C03650=1172.212,-91.528,-41.773,179.063,5.775,149.305
C03651=1172.217,-91.777,-41.762,179.061,5.775,149.306
C03652=1172.222,-92.027,-41.753,179.058,5.775,149.306
C03653=1172.228,-92.276,-41.743,179.057,5.775,149.307
C03654=1172.232,-92.527,-41.733,179.054,5.774,149.307
C03655=1172.238,-92.776,-41.723,179.052,5.773,149.308
C03656=1172.243,-93.026,-41.713,179.050,5.774,149.309
C03657=1172.249,-93.276,-41.704,179.048,5.773,149.309
C03658=1172.254,-93.525,-41.694,179.046,5.773,149.310
C03659=1172.259,-93.774,-41.684,179.043,5.773,149.310
C03660=1172.264,-94.025,-41.674,179.041,5.772,149.311
C03661=1172.270,-94.275,-41.664,179.039,5.772,149.312
C03662=1172.275,-94.524,-41.655,179.036,5.772,149.312
C03663=1172.281,-94.774,-41.645,179.035,5.772,149.313
C03664=1172.286,-95.023,-41.635,179.032,5.771,149.313
C03665=1172.291,-95.273,-41.625,179.030,5.771,149.314
C03666=1172.296,-95.524,-41.615,179.028,5.771,149.315
C03667=1172.301,-95.773,-41.606,179.026,5.770,149.315
C03668=1172.307,-96.023,-41.596,179.024,5.771,149.316
C03669=1172.312,-96.273,-41.587,179.021,5.770,149.316
C03670=1172.318,-96.522,-41.576,179.020,5.770,149.317
C03671=1172.323,-96.772,-41.568,179.017,5.770,149.318
C03672=1172.328,-97.021,-41.557,179.015,5.769,149.318
C03673=1172.333,-97.272,-41.548,179.013,5.769,149.319
C03674=1172.339,-97.522,-41.538,179.011,5.768,149.319
C03675=1172.344,-97.771,-41.529,179.009,5.769,149.320
C03676=1172.349,-98.021,-41.519,179.006,5.768,149.320
C03677=1172.354,-98.271,-41.510,179.004,5.768,149.321
C03678=1172.360,-98.520,-41.500,179.002,5.768,149.322
C03679=1172.365,-98.770,-41.490,179.000,5.767,149.322
C03680=1172.371,-99.020,-41.481,178.998,5.767,149.323
C03681=1172.376,-99.269,-41.471,178.995,5.767,149.323
C03682=1172.381,-99.520,-41.461,178.994,5.767,149.324
C03683=1172.386,-99.769,-41.451,178.991,5.766,149.324
C03684=1172.392,-100.019,-41.442,178.989,5.766,149.325
C03685=1172.397,-100.268,-41.432,178.987,5.766,149.326
C03686=1172.403,-100.519,-41.423,178.985,5.765,149.326
C03687=1172.408,-100.768,-41.414,178.983,5.765,149.327
C03688=1172.413,-101.018,-41.404,178.980,5.765,149.328
C03689=1172.418,-101.268,-41.395,178.979,5.765,149.328
C03690=1172.424,-101.517,-41.385,178.976,5.765,149.329
C03691=1172.430,-101.789,-41.374,178.974,5.764,149.329
C03692=1172.435,-102.061,-41.364,178.972,5.764,149.330
C03693=1172.441,-102.333,-41.354,178.969,5.764,149.331
C03694=1172.447,-102.605,-41.343,178.967,5.763,149.331
C03695=1172.452,-102.854,-41.334,178.965,5.764,149.332
C03696=1172.457,-103.104,-41.325,178.963,5.763,149.332
C03697=1172.463,-103.355,-41.315,178.960,5.762,149.333
C03698=1172.468,-103.604,-41.306,178.958,5.762,149.334
C03699=1172.473,-103.854,-41.296,178.956,5.762,149.334
C03700=1172.478,-104.103,-41.286,178.954,5.762,149.335
C03701=1172.484,-104.353,-41.278,178.952,5.761,149.335
C03702=1172.489,-104.603,-41.268,178.950,5.762,149.336
C03703=1172.494,-104.853,-41.258,178.948,5.761,149.336
C03704=1172.500,-105.103,-41.249,178.945,5.761,149.337
C03705=1172.505,-105.353,-41.240,178.943,5.761,149.338
C03706=1172.510,-105.602,-41.230,178.941,5.760,149.338
C03707=1172.516,-105.852,-41.221,178.939,5.760,149.339
C03708=1172.521,-106.102,-41.212,178.937,5.759,149.339
C03709=1172.526,-106.351,-41.202,178.935,5.760,149.340
C03710=1172.532,-106.601,-41.193,178.933,5.759,149.341
C03711=1172.537,-106.851,-41.184,178.930,5.760,149.341
C03712=1172.542,-107.100,-41.174,178.928,5.759,149.342
C03713=1172.548,-107.350,-41.165,178.927,5.759,149.342
C03714=1172.553,-107.600,-41.156,178.924,5.758,149.343
C03715=1172.558,-107.849,-41.146,178.922,5.758,149.343
C03716=1172.564,-108.100,-41.137,178.920,5.758,149.344
C03717=1172.569,-108.350,-41.128,178.918,5.757,149.345
C03718=1172.574,-108.599,-41.119,178.915,5.758,149.345
C03719=1172.580,-108.849,-41.109,178.913,5.757,149.346
C03720=1172.585,-109.099,-41.100,178.912,5.757,149.346
C03721=1172.590,-109.349,-41.091,178.909,5.757,149.347
C03722=1172.595,-109.598,-41.082,178.907,5.757,149.347
C03723=1172.601,-109.848,-41.072,178.905,5.756,149.348
C03724=1172.606,-110.098,-41.063,178.903,5.756,149.349
C03725=1172.611,-110.348,-41.054,178.901,5.755,149.349
C03726=1172.617,-110.598,-41.045,178.899,5.756,149.350
C03727=1172.622,-110.847,-41.035,178.897,5.755,149.350
C03728=1172.627,-111.097,-41.026,178.894,5.755,149.351
C03729=1172.632,-111.347,-41.017,178.892,5.755,149.352
C03730=1172.638,-111.597,-41.008,178.890,5.754,149.352
C03731=1172.644,-111.846,-40.999,178.888,5.754,149.353
C03732=1172.649,-112.095,-40.990,178.886,5.754,149.353
C03733=1172.654,-112.345,-40.981,178.884,5.754,149.354
C03734=1172.660,-112.595,-40.971,178.882,5.753,149.354
C03735=1172.665,-112.845,-40.962,178.880,5.753,149.355
C03736=1172.670,-113.095,-40.953,178.877,5.753,149.356
C03737=1172.675,-113.345,-40.945,178.876,5.753,149.356
C03738=1172.681,-113.595,-40.935,178.873,5.753,149.357
C03739=1172.686,-113.844,-40.925,178.871,5.753,149.357
C03740=1172.691,-114.094,-40.917,178.869,5.752,149.358
C03741=1172.697,-114.344,-40.908,178.867,5.752,149.359
C03742=1172.702,-114.594,-40.899,178.865,5.751,149.359
C03743=1172.708,-114.843,-40.890,178.863,5.752,149.360
C03744=1172.713,-115.093,-40.881,178.861,5.751,149.360
C03745=1172.719,-115.343,-40.872,178.859,5.751,149.361
C03746=1172.724,-115.593,-40.863,178.856,5.751,149.361
C03747=1172.729,-115.843,-40.854,178.854,5.750,149.362
C03748=1172.735,-116.093,-40.845,178.853,5.750,149.362
C03749=1172.740,-116.342,-40.835,178.850,5.750,149.363
C03750=1172.745,-116.592,-40.826,178.848,5.750,149.364
C03751=1172.750,-116.842,-40.817,178.846,5.749,149.364
C03752=1172.756,-117.091,-40.809,178.844,5.749,149.365
C03753=1172.761,-117.341,-40.800,178.842,5.749,149.365
C03754=1172.766,-117.591,-40.791,178.840,5.749,149.366
C03755=1172.772,-117.841,-40.781,178.838,5.748,149.367
C03756=1172.777,-118.091,-40.772,178.836,5.748,149.367
C03757=1172.782,-118.341,-40.764,178.833,5.748,149.368
C03758=1172.787,-118.590,-40.755,178.832,5.748,149.368
C03759=1172.793,-118.840,-40.746,178.829,5.748,149.369
C03760=1172.798,-119.089,-40.737,178.827,5.748,149.369
C03761=1172.804,-119.339,-40.728,178.825,5.747,149.370
C03762=1172.809,-119.589,-40.719,178.823,5.747,149.371
C03763=1172.815,-119.839,-40.710,178.821,5.746,149.371
C03764=1172.820,-120.089,-40.701,178.819,5.746,149.372
C03765=1172.825,-120.339,-40.692,178.817,5.746,149.372
C03766=1172.831,-120.588,-40.684,178.815,5.746,149.373
C03767=1172.836,-120.838,-40.675,178.812,5.746,149.373
C03768=1172.841,-121.088,-40.666,178.811,5.746,149.374
C03769=1172.846,-121.338,-40.657,178.809,5.745,149.374
C03770=1172.852,-121.588,-40.649,178.807,5.745,149.375
C03771=1172.857,-121.838,-40.640,178.804,5.745,149.376
C03772=1172.863,-122.087,-40.631,178.803,5.745,149.376
C03773=1172.868,-122.337,-40.622,178.800,5.744,149.377
C03774=1172.873,-122.587,-40.613,178.798,5.744,149.377
C03775=1172.878,-122.837,-40.605,178.796,5.744,149.378
C03776=1172.883,-123.087,-40.596,178.794,5.744,149.379
C03777=1172.889,-123.336,-40.587,178.792,5.743,149.379
C03778=1172.894,-123.586,-40.578,178.790,5.743,149.380
C03779=1172.899,-123.835,-40.569,178.788,5.743,149.380
C03780=1172.906,-124.086,-40.561,178.786,5.743,149.381
C03781=1172.911,-124.336,-40.552,178.784,5.742,149.381
C03782=1172.917,-124.585,-40.543,178.782,5.743,149.382
C03783=1172.922,-124.835,-40.534,178.780,5.742,149.382
C03784=1172.927,-125.085,-40.525,178.778,5.742,149.383
C03785=1172.932,-125.335,-40.516,178.775,5.741,149.384
C03786=1172.938,-125.584,-40.508,178.774,5.741,149.384
C03787=1172.943,-125.834,-40.500,178.772,5.741,149.385
C03788=1172.948,-126.084,-40.491,178.770,5.741,149.385
C03789=1172.954,-126.334,-40.482,178.767,5.740,149.386
C03790=1172.959,-126.583,-40.473,178.766,5.740,149.386
C03791=1172.964,-126.833,-40.465,178.763,5.740,149.387
C03792=1172.969,-127.083,-40.457,178.761,5.740,149.387
C03793=1172.974,-127.333,-40.448,178.759,5.739,149.388
C03794=1172.980,-127.582,-40.439,178.757,5.740,149.389
C03795=1172.559,-127.594,-40.480,178.753,5.743,149.391
C03796=1172.553,-127.344,-40.488,178.756,5.743,149.390
C03797=1172.548,-127.094,-40.497,178.758,5.743,149.389
C03798=1172.543,-126.844,-40.506,178.760,5.744,149.389
C03799=1172.537,-126.595,-40.515,178.762,5.744,149.388
C03800=1172.532,-126.344,-40.523,178.764,5.744,149.388
C03801=1172.527,-126.094,-40.532,178.766,5.744,149.387
C03802=1172.521,-125.845,-40.541,178.768,5.745,149.386
C03803=1172.516,-125.595,-40.549,178.770,5.745,149.386
C03804=1172.511,-125.346,-40.558,178.772,5.746,149.385
C03805=1172.505,-125.096,-40.567,178.774,5.745,149.385
C03806=1172.500,-124.845,-40.575,178.776,5.746,149.384
C03807=1172.494,-124.596,-40.584,178.778,5.746,149.384
C03808=1172.489,-124.346,-40.593,178.781,5.746,149.383
C03809=1172.484,-124.096,-40.602,178.782,5.746,149.383
C03810=1172.479,-123.847,-40.610,178.784,5.747,149.382
C03811=1172.473,-123.597,-40.619,178.787,5.746,149.381
C03812=1172.468,-123.348,-40.628,178.789,5.747,149.381
C03813=1172.462,-123.097,-40.636,178.790,5.747,149.380
C03814=1172.457,-122.847,-40.645,178.793,5.748,149.380
C03815=1172.452,-122.597,-40.654,178.795,5.748,149.379
C03816=1172.447,-122.348,-40.663,178.797,5.748,149.379
C03817=1172.441,-122.098,-40.671,178.799,5.748,149.378
C03818=1172.436,-121.849,-40.680,178.801,5.749,149.377
C03819=1172.431,-121.599,-40.689,178.803,5.749,149.377
C03820=1172.425,-121.349,-40.698,178.805,5.749,149.376
C03821=1172.420,-121.099,-40.707,178.807,5.749,149.376
C03822=1172.415,-120.850,-40.715,178.809,5.750,149.375
C03823=1172.409,-120.600,-40.724,178.811,5.749,149.375
C03824=1172.404,-120.350,-40.733,178.813,5.750,149.374
C03825=1172.399,-120.100,-40.742,178.815,5.750,149.374
C03826=1172.394,-119.850,-40.751,178.818,5.750,149.373
C03827=1172.388,-119.600,-40.761,178.819,5.750,149.372
C03828=1172.382,-119.351,-40.769,178.822,5.751,149.372
C03829=1172.377,-119.101,-40.777,178.824,5.751,149.371
C03830=1172.372,-118.851,-40.786,178.826,5.752,149.371
C03831=1172.366,-118.601,-40.795,178.828,5.751,149.370
C03832=1172.361,-118.351,-40.804,178.830,5.752,149.370
C03833=1172.356,-118.102,-40.814,178.832,5.752,149.369
C03834=1172.351,-117.852,-40.822,178.834,5.752,149.368
C03835=1172.345,-117.603,-40.831,178.836,5.752,149.368
C03836=1172.340,-117.353,-40.840,178.838,5.753,149.367
C03837=1172.334,-117.103,-40.849,178.840,5.753,149.367
C03838=1172.329,-116.853,-40.858,178.842,5.753,149.366
C03839=1172.324,-116.603,-40.867,178.844,5.753,149.365
C03840=1172.319,-116.353,-40.876,178.847,5.754,149.365
C03841=1172.314,-116.103,-40.885,178.848,5.754,149.364
C03842=1172.308,-115.853,-40.894,178.851,5.754,149.364
C03843=1172.302,-115.604,-40.903,178.853,5.754,149.363
C03844=1172.297,-115.354,-40.912,178.855,5.755,149.363
C03845=1172.292,-115.104,-40.921,178.857,5.754,149.362
C03846=1172.287,-114.855,-40.930,178.859,5.755,149.362
C03847=1172.281,-114.604,-40.939,178.861,5.755,149.361
C03848=1172.275,-114.355,-40.948,178.863,5.755,149.360
C03849=1172.271,-114.105,-40.958,178.865,5.755,149.360
C03850=1172.265,-113.856,-40.967,178.868,5.756,149.359
C03851=1172.260,-113.606,-40.975,178.869,5.756,149.359
C03852=1172.254,-113.355,-40.985,178.872,5.756,149.358
C03853=1172.249,-113.106,-40.994,178.873,5.756,149.358
C03854=1172.243,-112.856,-41.002,178.876,5.757,149.357
C03855=1172.238,-112.607,-41.011,178.878,5.757,149.356
C03856=1172.233,-112.357,-41.022,178.880,5.757,149.356
C03857=1172.227,-112.107,-41.030,178.883,5.758,149.355
C03858=1172.222,-111.857,-41.039,178.884,5.758,149.355
C03859=1172.217,-111.608,-41.048,178.886,5.758,149.354
C03860=1172.211,-111.357,-41.058,178.888,5.758,149.353
C03861=1172.206,-111.108,-41.067,178.891,5.759,149.353
C03862=1172.201,-110.858,-41.076,178.893,5.758,149.352
C03863=1172.196,-110.608,-41.085,178.895,5.759,149.352
C03864=1172.190,-110.358,-41.095,178.897,5.759,149.351
C03865=1172.185,-110.108,-41.104,178.899,5.759,149.351
C03866=1172.180,-109.859,-41.112,178.901,5.759,149.350
C03867=1172.175,-109.609,-41.122,178.903,5.760,149.349
C03868=1172.169,-109.359,-41.132,178.906,5.761,149.349
C03869=1172.164,-109.109,-41.140,178.907,5.761,149.348
C03870=1172.159,-108.859,-41.149,178.910,5.761,149.348
C03871=1172.153,-108.610,-41.160,178.912,5.761,149.347
C03872=1172.148,-108.360,-41.168,178.914,5.761,149.346
C03873=1172.143,-108.110,-41.177,178.916,5.761,149.346
C03874=1172.137,-107.860,-41.187,178.918,5.762,149.345
C03875=1172.132,-107.611,-41.196,178.920,5.762,149.345
C03876=1172.127,-107.361,-41.205,178.922,5.762,149.344
C03877=1172.121,-107.111,-41.215,178.924,5.762,149.344
C03878=1172.116,-106.862,-41.224,178.927,5.763,149.343
C03879=1172.111,-106.612,-41.233,178.929,5.763,149.342
C03880=1172.105,-106.362,-41.243,178.931,5.763,149.342
C03881=1172.100,-106.112,-41.252,178.933,5.764,149.341
C03882=1172.095,-105.862,-41.261,178.935,5.763,149.341
C03883=1172.089,-105.612,-41.271,178.937,5.764,149.340
C03884=1172.084,-105.363,-41.280,178.939,5.764,149.339
C03885=1172.079,-105.113,-41.289,178.942,5.765,149.339
C03886=1172.073,-104.863,-41.299,178.943,5.765,149.339
C03887=1172.068,-104.614,-41.308,178.946,5.765,149.338
C03888=1172.063,-104.364,-41.317,178.948,5.766,149.337
C03889=1172.057,-104.114,-41.327,178.950,5.765,149.337
C03890=1172.052,-103.865,-41.336,178.952,5.766,149.336
C03891=1172.046,-103.614,-41.346,178.954,5.766,149.335
C03892=1172.042,-103.365,-41.356,178.957,5.766,149.335
C03893=1172.036,-103.115,-41.364,178.959,5.766,149.334
C03894=1172.031,-102.865,-41.374,178.961,5.767,149.334
C03895=1172.026,-102.616,-41.384,178.962,5.767,149.333
C03896=1172.020,-102.344,-41.394,178.965,5.767,149.333
C03897=1172.014,-102.072,-41.405,178.968,5.768,149.332
C03898=1172.008,-101.801,-41.414,178.970,5.768,149.331
C03899=1172.002,-101.529,-41.425,178.972,5.768,149.331
C03900=1171.997,-101.279,-41.435,178.974,5.769,149.330
C03901=1171.992,-101.029,-41.444,178.976,5.768,149.329
C03902=1171.986,-100.779,-41.453,178.979,5.769,149.329
C03903=1171.981,-100.529,-41.463,178.981,5.769,149.328
C03904=1171.976,-100.279,-41.472,178.983,5.769,149.328
C03905=1171.971,-100.030,-41.482,178.986,5.770,149.327
C03906=1171.965,-99.780,-41.491,178.987,5.770,149.327
C03907=1171.960,-99.530,-41.501,178.990,5.770,149.326
C03908=1171.955,-99.281,-41.510,178.991,5.770,149.325
C03909=1171.949,-99.031,-41.521,178.994,5.771,149.325
C03910=1171.944,-98.781,-41.529,178.996,5.771,149.324
C03911=1171.938,-98.532,-41.540,178.998,5.771,149.324
C03912=1171.933,-98.282,-41.549,179.001,5.772,149.323
C03913=1171.928,-98.032,-41.559,179.002,5.772,149.322
C03914=1171.923,-97.782,-41.569,179.005,5.772,149.322
C03915=1171.917,-97.532,-41.578,179.006,5.772,149.321
C03916=1171.913,-97.283,-41.588,179.009,5.772,149.321
C03917=1171.907,-97.033,-41.597,179.011,5.773,149.320
C03918=1171.902,-96.783,-41.607,179.013,5.773,149.319
C03919=1171.896,-96.533,-41.616,179.016,5.774,149.319
C03920=1171.891,-96.284,-41.626,179.018,5.773,149.318
C03921=1171.886,-96.033,-41.636,179.020,5.774,149.318
C03922=1171.880,-95.784,-41.646,179.022,5.775,149.317
C03923=1171.875,-95.534,-41.656,179.024,5.774,149.316
C03924=1171.869,-95.284,-41.665,179.026,5.775,149.316
C03925=1171.865,-95.035,-41.675,179.028,5.775,149.315
C03926=1171.859,-94.786,-41.685,179.031,5.775,149.315
C03927=1171.854,-94.536,-41.694,179.033,5.776,149.314
C03928=1171.849,-94.285,-41.705,179.035,5.776,149.314
C03929=1171.843,-94.035,-41.714,179.037,5.776,149.313
C03930=1171.838,-93.786,-41.724,179.039,5.776,149.312
C03931=1171.832,-93.536,-41.734,179.042,5.777,149.312
C03932=1171.827,-93.287,-41.743,179.044,5.777,149.311
C03933=1171.822,-93.037,-41.753,179.046,5.777,149.310
C03934=1171.817,-92.787,-41.764,179.048,5.778,149.310
C03935=1171.811,-92.537,-41.772,179.050,5.777,149.309
C03936=1171.806,-92.287,-41.783,179.052,5.778,149.309
C03937=1171.801,-92.038,-41.792,179.055,5.779,149.308
C03938=1171.795,-91.789,-41.802,179.057,5.779,149.308
C03939=1171.790,-91.538,-41.812,179.059,5.779,149.307
C03940=1171.785,-91.289,-41.822,179.061,5.779,149.306
C03941=1171.780,-91.039,-41.832,179.063,5.780,149.306
C03942=1171.774,-90.789,-41.842,179.066,5.780,149.305
C03943=1171.769,-90.540,-41.851,179.067,5.780,149.305
C03944=1171.764,-90.289,-41.862,179.070,5.780,149.304
C03945=1171.758,-90.040,-41.872,179.072,5.780,149.304
C03946=1171.753,-89.790,-41.881,179.074,5.781,149.303
C03947=1171.748,-89.540,-41.891,179.077,5.782,149.302
C03948=1171.743,-89.290,-41.902,179.079,5.781,149.302
C03949=1171.738,-89.041,-41.911,179.081,5.782,149.301
C03950=1171.732,-88.791,-41.922,179.084,5.782,149.300
C03951=1171.726,-88.541,-41.931,179.085,5.782,149.300
C03952=1171.722,-88.291,-41.941,179.088,5.783,149.299
C03953=1171.716,-88.042,-41.951,179.089,5.783,149.299
C03954=1171.711,-87.792,-41.961,179.092,5.783,149.298
C03955=1171.706,-87.543,-41.971,179.094,5.784,149.298
C03956=1171.701,-87.292,-41.981,179.096,5.783,149.297
C03957=1171.695,-87.043,-41.991,179.099,5.784,149.296
C03958=1171.689,-86.793,-42.001,179.101,5.784,149.296
C03959=1171.684,-86.544,-42.011,179.103,5.785,149.295
C03960=1171.679,-86.294,-42.022,179.106,5.785,149.294
C03961=1171.674,-86.044,-42.032,179.107,5.785,149.294
C03962=1171.668,-85.795,-42.042,179.110,5.785,149.293
C03963=1171.664,-85.544,-42.051,179.112,5.786,149.293
C03964=1171.658,-85.294,-42.061,179.114,5.786,149.292
C03965=1171.653,-85.045,-42.072,179.116,5.787,149.292
C03966=1171.647,-84.795,-42.082,179.119,5.787,149.291
C03967=1171.643,-84.545,-42.092,179.120,5.787,149.290
C03968=1171.637,-84.296,-42.102,179.123,5.787,149.290
C03969=1171.631,-84.046,-42.112,179.125,5.787,149.289
C03970=1171.626,-83.796,-42.123,179.127,5.788,149.289
C03971=1171.622,-83.547,-42.132,179.130,5.789,149.288
C03972=1171.616,-83.297,-42.143,179.132,5.788,149.287
C03973=1171.611,-83.047,-42.153,179.134,5.789,149.287
C03974=1171.605,-82.797,-42.163,179.137,5.789,149.286
C03975=1171.600,-82.547,-42.173,179.138,5.789,149.286
C03976=1171.595,-82.297,-42.183,179.141,5.790,149.285
C03977=1171.590,-82.048,-42.193,179.143,5.790,149.284
C03978=1171.584,-81.798,-42.203,179.145,5.790,149.284
C03979=1171.579,-81.548,-42.214,179.147,5.791,149.283
C03980=1171.573,-81.299,-42.224,179.149,5.790,149.283
C03981=1171.568,-81.049,-42.234,179.152,5.791,149.282
C03982=1171.564,-80.799,-42.244,179.154,5.792,149.281
C03983=1171.558,-80.550,-42.254,179.156,5.791,149.281
C03984=1171.552,-80.300,-42.265,179.158,5.792,149.280
C03985=1171.547,-80.050,-42.275,179.161,5.792,149.279
C03986=1171.542,-79.800,-42.285,179.163,5.792,149.279
C03987=1171.536,-79.551,-42.296,179.165,5.793,149.278
C03988=1171.532,-79.301,-42.307,179.168,5.794,149.278
C03989=1171.526,-79.051,-42.317,179.170,5.793,149.277
C03990=1171.521,-78.802,-42.327,179.172,5.794,149.277
C03991=1171.516,-78.552,-42.337,179.175,5.794,149.276
C03992=1171.510,-78.302,-42.348,179.176,5.794,149.275
C03993=1171.505,-78.052,-42.358,179.179,5.795,149.275
C03994=1171.500,-77.803,-42.368,179.181,5.796,149.274
C03995=1171.494,-77.553,-42.379,179.183,5.795,149.274
C03996=1171.489,-77.303,-42.389,179.185,5.796,149.273
C03997=1171.484,-77.053,-42.399,179.188,5.796,149.272
C03998=1171.479,-76.803,-42.410,179.190,5.796,149.272
C03999=1171.473,-76.554,-42.420,179.192,5.797,149.271
C04000=1171.468,-76.283,-42.432,179.195,5.797,149.270
C04001=1171.462,-76.012,-42.443,179.197,5.798,149.270
C04002=1171.456,-75.741,-42.454,179.199,5.798,149.269
C04003=1171.451,-75.469,-42.465,179.202,5.798,149.269
C04004=1171.445,-75.220,-42.476,179.204,5.799,149.268
C04005=1171.440,-74.971,-42.487,179.207,5.799,149.267
C04006=1171.435,-74.720,-42.497,179.209,5.799,149.267
C04007=1171.429,-74.471,-42.507,179.211,5.800,149.266
C04008=1171.424,-74.221,-42.518,179.214,5.800,149.265
C04009=1171.418,-73.971,-42.528,179.215,5.800,149.265
C04010=1171.414,-73.721,-42.539,179.218,5.800,149.264
C04011=1171.408,-73.472,-42.550,179.220,5.801,149.264
C04012=1171.403,-73.222,-42.560,179.222,5.801,149.263
C04013=1171.398,-72.972,-42.570,179.224,5.802,149.263
C04014=1171.392,-72.723,-42.581,179.227,5.802,149.262
C04015=1171.387,-72.473,-42.592,179.229,5.802,149.261
C04016=1171.382,-72.223,-42.602,179.231,5.802,149.261
C04017=1171.377,-71.973,-42.613,179.234,5.803,149.260
C04018=1171.371,-71.724,-42.624,179.236,5.803,149.260
C04019=1171.366,-71.474,-42.634,179.238,5.803,149.259
C04020=1171.361,-71.224,-42.644,179.240,5.804,149.258
C04021=1171.356,-70.974,-42.655,179.242,5.804,149.258
C04022=1171.351,-70.725,-42.666,179.245,5.804,149.257
C04023=1171.346,-70.475,-42.676,179.247,5.805,149.256
C04024=1171.340,-70.225,-42.687,179.250,5.806,149.256
C04025=1171.335,-69.976,-42.698,179.252,5.805,149.255
C04026=1171.330,-69.726,-42.708,179.254,5.806,149.255
C04027=1171.324,-69.476,-42.719,179.256,5.806,149.254
C04028=1171.319,-69.227,-42.730,179.259,5.806,149.253
C04029=1171.314,-68.977,-42.741,179.261,5.807,149.253
C04030=1171.308,-68.727,-42.751,179.263,5.807,149.252
C04031=1171.303,-68.477,-42.762,179.265,5.807,149.252
C04032=1171.298,-68.228,-42.773,179.268,5.808,149.251
C04033=1171.293,-67.978,-42.783,179.270,5.808,149.250
C04034=1171.287,-67.729,-42.794,179.273,5.809,149.250
C04035=1171.282,-67.478,-42.805,179.274,5.809,149.249
C04036=1171.276,-67.229,-42.815,179.277,5.809,149.249
C04037=1171.271,-66.979,-42.827,179.279,5.810,149.248
C04038=1171.266,-66.729,-42.837,179.281,5.810,149.247
C04039=1171.261,-66.480,-42.848,179.284,5.810,149.247
C04040=1171.256,-66.230,-42.858,179.286,5.811,149.246
C04041=1171.251,-65.981,-42.870,179.289,5.811,149.246
C04042=1171.245,-65.731,-42.880,179.290,5.811,149.245
C04043=1171.240,-65.480,-42.891,179.293,5.812,149.244
C04044=1171.235,-65.231,-42.902,179.295,5.812,149.244
C04045=1171.229,-64.981,-42.913,179.297,5.812,149.243
C04046=1171.225,-64.732,-42.924,179.300,5.812,149.242
C04047=1171.219,-64.482,-42.934,179.302,5.813,149.242
C04048=1171.214,-64.233,-42.945,179.305,5.814,149.241
C04049=1171.208,-63.983,-42.956,179.306,5.814,149.241
C04050=1171.203,-63.733,-42.967,179.309,5.814,149.240
C04051=1171.198,-63.483,-42.978,179.311,5.815,149.240
C04052=1171.193,-63.234,-42.989,179.313,5.814,149.239
C04053=1171.188,-62.984,-43.000,179.316,5.815,149.238
C04054=1171.182,-62.734,-43.011,179.318,5.816,149.238
C04055=1171.177,-62.484,-43.022,179.321,5.816,149.237
C04056=1171.172,-62.235,-43.033,179.322,5.816,149.237
C04057=1171.167,-61.985,-43.043,179.325,5.816,149.236
C04058=1171.162,-61.735,-43.054,179.327,5.817,149.235
C04059=1171.156,-61.486,-43.065,179.330,5.818,149.235
C04060=1171.151,-61.236,-43.077,179.331,5.818,149.234
C04061=1171.146,-60.986,-43.088,179.334,5.818,149.233
C04062=1171.141,-60.737,-43.098,179.337,5.818,149.233
C04063=1171.135,-60.487,-43.110,179.338,5.818,149.232
C04064=1171.130,-60.237,-43.121,179.341,5.819,149.232
C04065=1171.125,-59.988,-43.131,179.343,5.820,149.231
C04066=1171.119,-59.738,-43.143,179.346,5.820,149.230
C04067=1171.114,-59.488,-43.154,179.348,5.820,149.230
C04068=1171.109,-59.239,-43.165,179.350,5.820,149.229
C04069=1171.104,-58.988,-43.175,179.353,5.821,149.228
C04070=1171.098,-58.739,-43.187,179.355,5.822,149.228
C04071=1171.093,-58.489,-43.198,179.357,5.821,149.227
C04072=1171.088,-58.239,-43.209,179.359,5.822,149.227
C04073=1171.082,-57.990,-43.220,179.362,5.823,149.226
C04074=1171.078,-57.740,-43.232,179.365,5.823,149.225
C04075=1171.073,-57.490,-43.242,179.366,5.823,149.225
C04076=1171.067,-57.241,-43.254,179.369,5.823,149.224
C04077=1171.062,-56.991,-43.265,179.371,5.824,149.224
C04078=1171.057,-56.741,-43.276,179.374,5.825,149.223
C04079=1171.052,-56.492,-43.286,179.375,5.825,149.223
C04080=1171.046,-56.242,-43.298,179.378,5.825,149.222
C04081=1171.042,-55.992,-43.310,179.381,5.825,149.221
C04082=1171.036,-55.742,-43.321,179.383,5.826,149.221
C04083=1171.031,-55.493,-43.332,179.385,5.826,149.220
C04084=1171.026,-55.243,-43.343,179.387,5.827,149.220
C04085=1171.020,-54.993,-43.355,179.390,5.827,149.219
C04086=1171.015,-54.744,-43.365,179.392,5.827,149.218
C04087=1171.010,-54.494,-43.376,179.394,5.827,149.218
C04088=1171.005,-54.244,-43.388,179.397,5.828,149.217
C04089=1171.000,-53.995,-43.400,179.399,5.829,149.216
C04090=1170.994,-53.745,-43.410,179.402,5.829,149.216
C04091=1170.989,-53.495,-43.422,179.404,5.830,149.215
C04092=1170.984,-53.246,-43.433,179.406,5.829,149.215
C04093=1170.979,-52.996,-43.445,179.408,5.830,149.214
C04094=1170.974,-52.747,-43.456,179.411,5.831,149.213
C04095=1170.968,-52.496,-43.467,179.413,5.831,149.213
C04096=1170.963,-52.247,-43.478,179.415,5.831,149.212
C04097=1170.958,-51.998,-43.489,179.418,5.832,149.212
C04098=1170.952,-51.748,-43.501,179.420,5.832,149.211
C04099=1170.948,-51.498,-43.512,179.422,5.833,149.210
C04100=1170.942,-51.248,-43.524,179.424,5.832,149.210
C04101=1170.938,-50.998,-43.536,179.427,5.833,149.209
C04102=1170.931,-50.749,-43.546,179.429,5.834,149.208
C04103=1170.927,-50.499,-43.558,179.432,5.834,149.208
C04104=1170.921,-50.229,-43.571,179.434,5.835,149.207
C04105=1170.915,-49.958,-43.582,179.437,5.835,149.207
C04106=1170.910,-49.688,-43.595,179.440,5.836,149.206
C04107=1170.904,-49.417,-43.608,179.442,5.836,149.205
C04108=1170.899,-49.168,-43.619,179.444,5.836,149.205
C04109=1170.893,-48.918,-43.630,179.446,5.837,149.204
C04110=1170.889,-48.669,-43.642,179.449,5.837,149.203
C04111=1170.883,-48.419,-43.654,179.451,5.838,149.203
C04112=1170.878,-48.169,-43.666,179.454,5.838,149.202
C04113=1170.873,-47.920,-43.676,179.456,5.838,149.202
C04114=1170.867,-47.670,-43.688,179.458,5.839,149.201
C04115=1170.862,-47.420,-43.700,179.460,5.839,149.200
C04116=1170.857,-47.170,-43.712,179.463,5.840,149.200
C04117=1170.852,-46.921,-43.723,179.465,5.839,149.199
C04118=1170.846,-46.671,-43.734,179.467,5.840,149.199
C04119=1170.841,-46.421,-43.745,179.470,5.841,149.198
C04120=1170.836,-46.172,-43.758,179.472,5.841,149.197
C04121=1170.831,-45.922,-43.769,179.475,5.842,149.197
C04122=1170.826,-45.672,-43.781,179.477,5.842,149.196
C04123=1170.821,-45.422,-43.793,179.479,5.842,149.196
C04124=1170.815,-45.173,-43.803,179.482,5.843,149.195
C04125=1170.810,-44.923,-43.815,179.484,5.844,149.194
C04126=1170.805,-44.674,-43.827,179.487,5.844,149.194
C04127=1170.800,-44.424,-43.839,179.489,5.844,149.193
C04128=1170.794,-44.174,-43.850,179.491,5.844,149.192
C04129=1170.790,-43.924,-43.862,179.494,5.845,149.192
C04130=1170.784,-43.674,-43.874,179.496,5.846,149.191
C04131=1170.778,-43.425,-43.885,179.498,5.846,149.191
C04132=1170.774,-43.176,-43.896,179.501,5.846,149.190
C04133=1170.768,-42.926,-43.908,179.503,5.846,149.189
C04134=1170.763,-42.676,-43.920,179.505,5.847,149.189
C04135=1170.758,-42.427,-43.932,179.507,5.848,149.188
C04136=1170.753,-42.177,-43.944,179.510,5.848,149.188
C04137=1170.748,-41.927,-43.955,179.513,5.849,149.187
C04138=1170.743,-41.677,-43.967,179.515,5.849,149.186
C04139=1170.737,-41.427,-43.979,179.517,5.849,149.186
C04140=1170.732,-41.178,-43.990,179.520,5.849,149.185
C04141=1170.727,-40.928,-44.002,179.522,5.850,149.184
C04142=1170.721,-40.679,-44.015,179.525,5.851,149.184
C04143=1170.717,-40.429,-44.026,179.527,5.851,149.183
C04144=1170.711,-40.180,-44.038,179.529,5.851,149.183
C04145=1170.706,-39.930,-44.050,179.531,5.852,149.182
C04146=1170.700,-39.680,-44.062,179.534,5.852,149.181
C04147=1170.696,-39.431,-44.074,179.536,5.853,149.181
C04148=1170.691,-39.181,-44.085,179.539,5.854,149.180
C04149=1170.685,-38.931,-44.097,179.541,5.854,149.180
C04150=1170.681,-38.681,-44.109,179.543,5.854,149.179
C04151=1170.675,-38.432,-44.121,179.545,5.854,149.178
C04152=1170.670,-38.182,-44.133,179.548,5.855,149.178
C04153=1170.664,-37.933,-44.145,179.550,5.856,149.177
C04154=1170.659,-37.683,-44.156,179.553,5.856,149.176
C04155=1170.654,-37.434,-44.168,179.556,5.857,149.176
C04156=1170.649,-37.184,-44.180,179.558,5.857,149.175
C04157=1170.643,-36.934,-44.192,179.560,5.857,149.175
C04158=1170.638,-36.684,-44.204,179.562,5.858,149.174
C04159=1170.633,-36.435,-44.216,179.565,5.858,149.173
C04160=1170.628,-36.185,-44.228,179.567,5.859,149.173
C04161=1170.623,-35.935,-44.240,179.570,5.859,149.172
C04162=1170.617,-35.686,-44.252,179.572,5.860,149.172
C04163=1170.613,-35.436,-44.264,179.574,5.861,149.171
C04164=1170.607,-35.186,-44.276,179.576,5.860,149.170
C04165=1170.602,-34.937,-44.288,179.579,5.861,149.170
C04166=1170.597,-34.687,-44.300,179.581,5.862,149.169
C04167=1170.591,-34.437,-44.312,179.584,5.862,149.169
C04168=1170.586,-34.188,-44.325,179.587,5.862,149.168
C04169=1170.582,-33.938,-44.336,179.589,5.863,149.167
C04170=1170.576,-33.689,-44.349,179.591,5.864,149.167
C04171=1170.571,-33.439,-44.360,179.593,5.864,149.166
C04172=1170.566,-33.189,-44.372,179.596,5.864,149.165
C04173=1170.560,-32.939,-44.385,179.598,5.865,149.165
C04174=1170.555,-32.690,-44.397,179.601,5.865,149.164
C04175=1170.550,-32.440,-44.409,179.603,5.866,149.164
C04176=1170.545,-32.191,-44.421,179.605,5.867,149.163
C04177=1170.540,-31.941,-44.433,179.608,5.867,149.162
C04178=1170.535,-31.691,-44.445,179.610,5.867,149.162
C04179=1170.529,-31.441,-44.457,179.612,5.868,149.161
C04180=1170.524,-31.192,-44.470,179.615,5.868,149.161
C04181=1170.519,-30.941,-44.482,179.618,5.868,149.160
C04182=1170.514,-30.692,-44.495,179.620,5.869,149.159
C04183=1170.509,-30.442,-44.506,179.622,5.870,149.159
C04184=1170.504,-30.193,-44.519,179.625,5.870,149.158
C04185=1170.498,-29.943,-44.531,179.627,5.871,149.158
C04186=1170.494,-29.694,-44.543,179.629,5.871,149.157
C04187=1170.488,-29.444,-44.555,179.632,5.871,149.156
C04188=1170.483,-29.195,-44.567,179.634,5.872,149.156
C04189=1170.478,-28.945,-44.580,179.636,5.873,149.155
C04190=1170.473,-28.695,-44.592,179.639,5.873,149.155
C04191=1170.468,-28.446,-44.604,179.642,5.873,149.154
C04192=1170.462,-28.196,-44.616,179.644,5.874,149.153
C04193=1170.458,-27.946,-44.629,179.647,5.875,149.153
C04194=1170.452,-27.696,-44.641,179.649,5.875,149.152
C04195=1170.447,-27.447,-44.654,179.651,5.875,149.151
C04196=1170.442,-27.198,-44.666,179.653,5.876,149.151
C04197=1170.436,-26.948,-44.678,179.656,5.876,149.150
C04198=1170.431,-26.698,-44.691,179.658,5.877,149.150
C04199=1170.426,-26.448,-44.703,179.661,5.877,149.149
C04200=1170.421,-26.199,-44.715,179.663,5.878,149.148
C04201=1170.416,-25.950,-44.728,179.666,5.879,149.148
C04202=1170.411,-25.699,-44.740,179.668,5.879,149.147
C04203=1170.406,-25.450,-44.753,179.671,5.880,149.147
C04204=1170.401,-25.200,-44.765,179.673,5.880,149.146
C04205=1170.395,-24.951,-44.777,179.675,5.880,149.145
C04206=1170.390,-24.701,-44.790,179.678,5.881,149.145
C04207=1170.385,-24.452,-44.803,179.680,5.881,149.144
C04208=1170.380,-24.182,-44.815,179.682,5.882,149.144
C04209=1170.374,-23.912,-44.830,179.685,5.882,149.143
C04210=1170.368,-23.642,-44.842,179.688,5.884,149.142
C04211=1170.363,-23.372,-44.856,179.691,5.884,149.141
C04212=1170.357,-23.123,-44.869,179.693,5.884,149.141
C04213=1170.352,-22.873,-44.882,179.695,5.885,149.140
C04214=1170.347,-22.623,-44.894,179.698,5.885,149.140
C04215=1170.342,-22.373,-44.907,179.700,5.886,149.139
C04216=1170.337,-22.124,-44.919,179.703,5.886,149.138
C04217=1170.332,-21.875,-44.932,179.705,5.887,149.138
C04218=1170.326,-21.625,-44.944,179.708,5.887,149.137
C04219=1170.321,-21.375,-44.956,179.710,5.888,149.137
C04220=1170.317,-21.125,-44.969,179.712,5.889,149.136
C04221=1170.312,-20.876,-44.982,179.715,5.889,149.135
C04222=1170.305,-20.626,-44.994,179.718,5.890,149.135
C04223=1170.300,-20.376,-45.007,179.720,5.890,149.134
C04224=1170.295,-20.127,-45.020,179.723,5.891,149.134
C04225=1170.291,-19.877,-45.033,179.725,5.891,149.133
C04226=1170.286,-19.628,-45.045,179.727,5.891,149.132
C04227=1170.280,-19.378,-45.058,179.729,5.892,149.132
C04228=1170.274,-19.128,-45.070,179.732,5.893,149.131
C04229=1170.270,-18.878,-45.083,179.734,5.893,149.131
C04230=1170.265,-18.629,-45.096,179.737,5.893,149.130
C04231=1170.259,-18.380,-45.108,179.739,5.894,149.129
C04232=1170.254,-18.130,-45.121,179.742,5.895,149.129
C04233=1170.250,-17.880,-45.134,179.744,5.895,149.128
C04234=1170.244,-17.631,-45.147,179.747,5.896,149.128
C04235=1170.239,-17.381,-45.160,179.749,5.896,149.127
C04236=1170.233,-17.131,-45.172,179.752,5.897,149.126
C04237=1170.229,-16.881,-45.185,179.754,5.898,149.126
C04238=1170.223,-16.632,-45.198,179.757,5.898,149.125
C04239=1170.218,-16.382,-45.210,179.759,5.899,149.124
C04240=1170.213,-16.133,-45.223,179.762,5.899,149.124
C04241=1170.208,-15.883,-45.236,179.764,5.900,149.123
C04242=1170.203,-15.634,-45.249,179.766,5.901,149.123
C04243=1170.197,-15.384,-45.262,179.769,5.901,149.122
C04244=1170.193,-15.134,-45.275,179.771,5.901,149.121
C04245=1170.188,-14.885,-45.287,179.773,5.902,149.121
C04246=1170.182,-14.635,-45.301,179.776,5.902,149.120
C04247=1170.177,-14.386,-45.313,179.778,5.903,149.120
C04248=1170.172,-14.136,-45.326,179.781,5.903,149.119
C04249=1170.167,-13.887,-45.339,179.783,5.904,149.118
C04250=1170.161,-13.637,-45.352,179.786,5.905,149.118
C04251=1170.157,-13.387,-45.365,179.788,5.905,149.117
C04252=1170.151,-13.138,-45.377,179.791,5.906,149.117
C04253=1170.146,-12.888,-45.391,179.793,5.906,149.116
C04254=1170.141,-12.638,-45.404,179.796,5.907,149.115
C04255=1170.136,-12.389,-45.416,179.798,5.908,149.115
C04256=1170.131,-12.139,-45.429,179.801,5.908,149.114
C04257=1170.126,-11.890,-45.443,179.803,5.909,149.114
C04258=1170.121,-11.640,-45.456,179.806,5.909,149.113
C04259=1170.116,-11.391,-45.468,179.808,5.910,149.112
C04260=1170.110,-11.141,-45.482,179.810,5.911,149.112
C04261=1170.105,-10.891,-45.494,179.813,5.911,149.111
C04262=1170.099,-10.642,-45.508,179.816,5.912,149.110
C04263=1170.095,-10.392,-45.521,179.818,5.912,149.110
C04264=1170.090,-10.142,-45.533,179.821,5.913,149.109
C04265=1170.084,-9.892,-45.547,179.823,5.914,149.109
C04266=1170.080,-9.643,-45.560,179.825,5.914,149.108
C04267=1170.075,-9.394,-45.573,179.828,5.915,149.107
C04268=1170.069,-9.144,-45.586,179.830,5.915,149.107
C04269=1170.064,-8.894,-45.599,179.833,5.916,149.106
C04270=1170.059,-8.644,-45.612,179.835,5.917,149.106
C04271=1170.054,-8.395,-45.626,179.838,5.917,149.105
C04272=1170.049,-8.146,-45.638,179.840,5.918,149.104
C04273=1170.044,-7.896,-45.652,179.842,5.918,149.104
C04274=1170.039,-7.646,-45.665,179.845,5.919,149.103
C04275=1170.033,-7.396,-45.678,179.848,5.919,149.103
C04276=1170.028,-7.147,-45.691,179.850,5.920,149.102
C04277=1170.023,-6.898,-45.705,179.853,5.921,149.101
C04278=1170.018,-6.648,-45.718,179.855,5.921,149.101
C04279=1170.013,-6.398,-45.730,179.857,5.922,149.100
C04280=1170.008,-6.149,-45.744,179.860,5.922,149.100
C04281=1170.003,-5.899,-45.757,179.862,5.923,149.099
C04282=1169.998,-5.649,-45.771,179.865,5.924,149.098
C04283=1169.993,-5.400,-45.784,179.868,5.924,149.098
C04284=1169.987,-5.151,-45.797,179.870,5.925,149.097
C04285=1169.982,-4.901,-45.810,179.872,5.925,149.097
C04286=1169.977,-4.651,-45.823,179.875,5.926,149.096
C04287=1169.972,-4.402,-45.837,179.877,5.927,149.095
C04288=1169.966,-4.152,-45.850,179.880,5.927,149.095
C04289=1169.962,-3.902,-45.863,179.882,5.928,149.094
C04290=1169.956,-3.653,-45.877,179.885,5.928,149.094
C04291=1169.952,-3.403,-45.890,179.887,5.929,149.093
C04292=1169.946,-3.154,-45.904,179.890,5.930,149.092
C04293=1169.942,-2.904,-45.917,179.892,5.930,149.092
C04294=1169.936,-2.654,-45.930,179.894,5.931,149.091
C04295=1169.931,-2.405,-45.944,179.897,5.931,149.091
C04296=1169.926,-2.155,-45.957,179.900,5.932,149.090
C04297=1169.921,-1.906,-45.971,179.902,5.933,149.089
C04298=1169.916,-1.656,-45.984,179.905,5.933,149.089
C04299=1169.911,-1.406,-45.997,179.907,5.934,149.088
C04300=1169.906,-1.157,-46.011,179.909,5.934,149.088
C04301=1169.900,-0.907,-46.024,179.912,5.935,149.087
C04302=1169.895,-0.658,-46.038,179.914,5.936,149.086
C04303=1169.890,-0.408,-46.051,179.917,5.936,149.086
C04304=1169.885,-0.159,-46.065,179.919,5.937,149.085
C04305=1169.880,0.091,-46.078,179.922,5.937,149.085
C04306=1169.875,0.340,-46.092,179.924,5.938,149.084
C04307=1169.869,0.591,-46.106,179.927,5.940,149.083
C04308=1169.865,0.839,-46.119,179.930,5.940,149.083
C04309=1169.859,1.090,-46.132,179.932,5.940,149.082
C04310=1169.854,1.339,-46.146,179.935,5.941,149.082
C04311=1169.849,1.589,-46.159,179.937,5.942,149.081
C04312=1169.844,1.858,-46.174,179.940,5.942,149.080
C04313=1169.838,2.127,-46.189,179.942,5.943,149.080
C04314=1169.832,2.396,-46.204,179.945,5.943,149.079
C04315=1169.827,2.666,-46.218,179.948,5.945,149.078
C04316=1169.822,2.916,-46.232,179.951,5.945,149.078
C04317=1169.817,3.165,-46.246,179.953,5.946,149.077
C04318=1169.812,3.415,-46.259,179.955,5.947,149.076
C04319=1169.807,3.664,-46.273,179.958,5.947,149.076
C04320=1169.802,3.914,-46.286,179.960,5.948,149.075
C04321=1169.796,4.163,-46.300,179.963,5.948,149.075
C04322=1169.792,4.412,-46.314,179.965,5.949,149.074
C04323=1169.787,4.663,-46.327,179.968,5.950,149.074
C04324=1169.781,4.912,-46.341,179.970,5.950,149.073
C04325=1169.776,5.162,-46.354,179.973,5.951,149.072
C04326=1169.772,5.411,-46.369,179.975,5.951,149.072
C04327=1169.766,5.660,-46.382,179.977,5.952,149.071
C04328=1169.761,5.911,-46.396,179.980,5.953,149.071
C04329=1169.756,6.159,-46.409,179.983,5.953,149.070
C04330=1169.751,6.409,-46.424,179.985,5.955,149.069
C04331=1169.746,6.659,-46.438,179.988,5.955,149.069
C04332=1169.740,6.909,-46.451,179.990,5.956,149.068
C04333=1169.736,7.158,-46.465,179.993,5.956,149.068
C04334=1169.731,7.408,-46.479,179.996,5.957,149.067
C04335=1169.725,7.657,-46.492,179.998,5.958,149.066
C04336=1169.720,7.907,-46.506,-180.000,5.958,149.066
C04337=1169.715,8.157,-46.521,-179.997,5.959,149.065
C04338=1169.710,8.405,-46.534,-179.995,5.960,149.065
C04339=1169.705,8.656,-46.548,-179.992,5.960,149.064
C04340=1169.700,8.905,-46.562,-179.990,5.961,149.063
C04341=1169.695,9.154,-46.576,-179.987,5.961,149.063
C04342=1169.690,9.404,-46.590,-179.985,5.963,149.062
C04343=1169.685,9.654,-46.604,-179.982,5.963,149.062
C04344=1169.680,9.903,-46.617,-179.979,5.964,149.061
C04345=1169.675,10.153,-46.631,-179.977,5.965,149.060
C04346=1169.670,10.403,-46.646,-179.974,5.965,149.060
C04347=1169.664,10.652,-46.659,-179.972,5.966,149.059
C04348=1169.659,10.901,-46.674,-179.970,5.967,149.059
C04349=1169.654,11.151,-46.688,-179.967,5.967,149.058
C04350=1169.648,11.401,-46.701,-179.965,5.968,149.057
C04351=1169.643,11.650,-46.715,-179.962,5.968,149.057
C04352=1169.639,11.900,-46.729,-179.959,5.970,149.056
C04353=1169.634,12.149,-46.743,-179.957,5.970,149.056
C04354=1169.629,12.398,-46.757,-179.954,5.971,149.055
C04355=1169.624,12.648,-46.772,-179.952,5.972,149.055
C04356=1169.619,12.898,-46.786,-179.949,5.972,149.054
C04357=1169.613,13.147,-46.800,-179.947,5.973,149.053
C04358=1169.608,13.397,-46.814,-179.944,5.974,149.053
C04359=1169.603,13.646,-46.828,-179.942,5.974,149.052
C04360=1169.598,13.897,-46.842,-179.940,5.975,149.052
C04361=1169.592,14.146,-46.856,-179.936,5.976,149.051
C04362=1169.587,14.395,-46.870,-179.934,5.977,149.050
C04363=1169.583,14.645,-46.884,-179.932,5.977,149.050
C04364=1169.578,14.895,-46.899,-179.929,5.978,149.049
C04365=1169.573,15.145,-46.913,-179.927,5.979,149.049
C04366=1169.567,15.394,-46.927,-179.924,5.979,149.048
C04367=1169.563,15.643,-46.941,-179.921,5.980,149.047
C04368=1169.558,15.893,-46.955,-179.919,5.980,149.047
C04369=1169.553,16.142,-46.969,-179.916,5.982,149.046
C04370=1169.547,16.391,-46.983,-179.914,5.983,149.046
C04371=1169.542,16.641,-46.997,-179.911,5.983,149.045
C04372=1169.537,16.891,-47.012,-179.909,5.984,149.044
C04373=1169.533,17.140,-47.027,-179.906,5.984,149.044
C04374=1169.527,17.390,-47.041,-179.904,5.985,149.043
C04375=1169.522,17.639,-47.055,-179.902,5.986,149.043
C04376=1169.517,17.889,-47.070,-179.898,5.987,149.042
C04377=1169.512,18.138,-47.084,-179.896,5.988,149.042
C04378=1169.507,18.388,-47.098,-179.894,5.988,149.041
C04379=1169.502,18.638,-47.112,-179.891,5.989,149.040
C04380=1169.497,18.887,-47.127,-179.889,5.990,149.040
C04381=1169.491,19.136,-47.141,-179.886,5.990,149.039
C04382=1169.486,19.386,-47.155,-179.884,5.991,149.039
C04383=1169.482,19.635,-47.170,-179.881,5.992,149.038
C04384=1169.477,19.885,-47.184,-179.878,5.993,149.037
C04385=1169.472,20.135,-47.198,-179.876,5.994,149.037
C04386=1169.467,20.384,-47.213,-179.873,5.994,149.036
C04387=1169.461,20.633,-47.227,-179.871,5.995,149.036
C04388=1169.456,20.883,-47.241,-179.868,5.995,149.035
C04389=1169.451,21.133,-47.257,-179.865,5.997,149.034
C04390=1169.446,21.382,-47.271,-179.863,5.997,149.034
C04391=1169.441,21.632,-47.285,-179.860,5.998,149.033
C04392=1169.436,21.882,-47.299,-179.858,5.999,149.033
C04393=1169.431,22.131,-47.314,-179.856,5.999,149.032
C04394=1169.426,22.380,-47.329,-179.853,6.000,149.032
C04395=1169.421,22.629,-47.343,-179.850,6.001,149.031
C04396=1169.415,22.879,-47.357,-179.847,6.002,149.030
C04397=1169.410,23.129,-47.372,-179.845,6.003,149.030
C04398=1169.406,23.378,-47.387,-179.843,6.003,149.029
C04399=1169.401,23.628,-47.401,-179.841,6.004,149.029
C04400=1169.396,23.878,-47.415,-179.838,6.005,149.028
C04401=1169.391,24.127,-47.430,-179.835,6.006,149.027
C04402=1169.385,24.377,-47.445,-179.832,6.007,149.027
C04403=1169.380,24.627,-47.459,-179.830,6.007,149.026
C04404=1169.376,24.876,-47.474,-179.828,6.008,149.026
C04405=1169.371,25.125,-47.489,-179.825,6.008,149.025
C04406=1169.366,25.375,-47.503,-179.822,6.010,149.025
C04407=1169.360,25.624,-47.518,-179.820,6.011,149.024
C04408=1169.355,25.873,-47.532,-179.817,6.011,149.023
C04409=1169.350,26.123,-47.547,-179.815,6.012,149.023
C04410=1169.345,26.372,-47.562,-179.812,6.012,149.022
C04411=1169.340,26.622,-47.577,-179.810,6.013,149.022
C04412=1169.335,26.872,-47.591,-179.807,6.015,149.021
C04413=1169.330,27.121,-47.606,-179.804,6.015,149.020
C04414=1169.325,27.371,-47.620,-179.802,6.016,149.020
C04415=1169.320,27.620,-47.636,-179.799,6.016,149.019
C04416=1169.314,27.889,-47.651,-179.797,6.018,149.019
C04417=1169.309,28.158,-47.667,-179.794,6.018,149.018
C04418=1169.303,28.427,-47.683,-179.791,6.019,149.017
C04419=1169.298,28.696,-47.699,-179.788,6.020,149.017
C04420=1169.293,28.946,-47.714,-179.786,6.021,149.016
C04421=1169.288,29.195,-47.729,-179.783,6.022,149.015
C04422=1169.283,29.444,-47.743,-179.781,6.022,149.015
C04423=1169.278,29.694,-47.758,-179.778,6.024,149.014
C04424=1169.273,29.944,-47.773,-179.775,6.024,149.014
C04425=1169.268,30.193,-47.788,-179.773,6.025,149.013
C04426=1169.262,30.443,-47.803,-179.770,6.026,149.013
C04427=1169.258,30.692,-47.818,-179.768,6.026,149.012
C04428=1169.253,30.942,-47.832,-179.765,6.028,149.011
C04429=1169.247,31.191,-47.848,-179.762,6.028,149.011
C04430=1169.242,31.441,-47.862,-179.760,6.029,149.010
C04431=1169.238,31.690,-47.877,-179.758,6.030,149.010
C04432=1169.232,31.940,-47.892,-179.755,6.031,149.009
C04433=1169.227,32.189,-47.907,-179.752,6.032,149.008
C04434=1169.223,32.438,-47.922,-179.750,6.033,149.008
C04435=1169.217,32.688,-47.937,-179.747,6.033,149.007
C04436=1169.212,32.937,-47.952,-179.745,6.034,149.007
C04437=1169.207,33.187,-47.967,-179.742,6.035,149.006
C04438=1169.202,33.436,-47.982,-179.739,6.036,149.006
C04439=1169.197,33.686,-47.998,-179.737,6.036,149.005
C04440=1169.192,33.936,-48.012,-179.734,6.037,149.004
C04441=1169.188,34.185,-48.027,-179.732,6.039,149.004
C04442=1169.182,34.434,-48.043,-179.729,6.039,149.003
C04443=1169.177,34.684,-48.057,-179.727,6.040,149.003
C04444=1169.172,34.934,-48.072,-179.724,6.040,149.002
C04445=1169.167,35.183,-48.087,-179.721,6.042,149.002
C04446=1169.162,35.433,-48.102,-179.719,6.043,149.001
C04447=1169.157,35.682,-48.117,-179.716,6.043,149.000
C04448=1169.152,35.931,-48.133,-179.714,6.044,149.000
C04449=1169.147,36.180,-48.148,-179.711,6.045,148.999
C04450=1169.142,36.431,-48.163,-179.709,6.046,148.999
C04451=1169.137,36.680,-48.178,-179.706,6.047,148.998
C04452=1169.132,36.929,-48.194,-179.704,6.047,148.998
C04453=1169.127,37.179,-48.209,-179.701,6.049,148.997
C04454=1169.121,37.429,-48.223,-179.698,6.049,148.996
C04455=1169.117,37.678,-48.238,-179.696,6.050,148.996
C04456=1169.111,37.927,-48.254,-179.693,6.051,148.995
C04457=1169.107,38.176,-48.269,-179.690,6.052,148.995
C04458=1169.102,38.426,-48.285,-179.688,6.053,148.994
C04459=1169.097,38.676,-48.299,-179.686,6.054,148.994
C04460=1169.092,38.925,-48.315,-179.683,6.054,148.993
C04461=1169.086,39.175,-48.330,-179.680,6.056,148.993
C04462=1169.082,39.424,-48.345,-179.678,6.056,148.992
C04463=1169.076,39.673,-48.361,-179.675,6.057,148.991
C04464=1169.072,39.923,-48.376,-179.672,6.058,148.991
C04465=1169.067,40.173,-48.391,-179.670,6.059,148.990
C04466=1169.061,40.423,-48.407,-179.667,6.060,148.990
C04467=1169.056,40.672,-48.422,-179.665,6.060,148.989
C04468=1169.051,40.921,-48.437,-179.662,6.062,148.989
C04469=1169.046,41.170,-48.452,-179.659,6.062,148.988
C04470=1169.042,41.420,-48.468,-179.657,6.063,148.987
C04471=1169.036,41.670,-48.484,-179.655,6.064,148.987
C04472=1169.032,41.919,-48.499,-179.652,6.065,148.986
C04473=1169.026,42.168,-48.515,-179.649,6.066,148.986
C04474=1169.021,42.418,-48.531,-179.647,6.066,148.985
C04475=1169.017,42.667,-48.546,-179.644,6.068,148.984
C04476=1169.011,42.917,-48.561,-179.641,6.069,148.984
C04477=1169.006,43.166,-48.577,-179.639,6.069,148.983
C04478=1169.001,43.415,-48.592,-179.636,6.071,148.983
C04479=1168.997,43.665,-48.608,-179.634,6.072,148.982
C04480=1168.991,43.915,-48.623,-179.631,6.072,148.982
C04481=1168.987,44.164,-48.638,-179.629,6.073,148.981
C04482=1168.981,44.413,-48.654,-179.626,6.074,148.980
C04483=1168.976,44.663,-48.670,-179.623,6.075,148.980
C04484=1168.972,44.912,-48.685,-179.621,6.076,148.979
C04485=1168.966,45.162,-48.700,-179.618,6.077,148.979
C04486=1168.961,45.411,-48.716,-179.615,6.078,148.978
C04487=1168.956,45.661,-48.732,-179.613,6.079,148.978
C04488=1168.952,45.910,-48.747,-179.610,6.080,148.977
C04489=1168.946,46.160,-48.762,-179.607,6.080,148.976
C04490=1168.941,46.410,-48.778,-179.605,6.081,148.976
C04491=1168.937,46.659,-48.793,-179.603,6.082,148.975
C04492=1168.931,46.908,-48.809,-179.600,6.083,148.975
C04493=1168.926,47.158,-48.825,-179.597,6.084,148.974
C04494=1168.921,47.407,-48.841,-179.595,6.085,148.974
C04495=1168.916,47.657,-48.857,-179.592,6.086,148.973
C04496=1168.911,47.906,-48.872,-179.590,6.087,148.973
C04497=1168.907,48.156,-48.888,-179.587,6.087,148.972
C04498=1168.901,48.405,-48.903,-179.584,6.089,148.972
C04499=1168.896,48.655,-48.919,-179.582,6.090,148.971
C04500=1168.891,48.904,-48.936,-179.580,6.090,148.970
C04501=1168.887,49.153,-48.951,-179.576,6.092,148.970
C04502=1168.881,49.403,-48.966,-179.574,6.093,148.969
C04503=1168.877,49.653,-48.982,-179.572,6.093,148.969
C04504=1168.871,49.902,-48.998,-179.569,6.095,148.968
C04505=1168.866,50.151,-49.014,-179.566,6.095,148.968
C04506=1168.862,50.401,-49.029,-179.564,6.096,148.967
C04507=1168.857,50.650,-49.045,-179.561,6.097,148.966
C04508=1168.852,50.899,-49.061,-179.558,6.098,148.966
C04509=1168.847,51.149,-49.077,-179.556,6.099,148.965
C04510=1168.841,51.398,-49.093,-179.553,6.100,148.965
C04511=1168.837,51.649,-49.109,-179.551,6.101,148.964
C04512=1168.832,51.897,-49.125,-179.548,6.102,148.964
C04513=1168.826,52.147,-49.141,-179.545,6.103,148.963
C04514=1168.822,52.396,-49.156,-179.543,6.104,148.962
C04515=1168.817,52.645,-49.172,-179.540,6.105,148.962
C04516=1168.812,52.895,-49.188,-179.537,6.106,148.961
C04517=1168.807,53.145,-49.204,-179.535,6.107,148.961
C04518=1168.802,53.394,-49.220,-179.532,6.108,148.960
C04519=1168.797,53.644,-49.236,-179.530,6.109,148.960
C04520=1168.791,53.912,-49.253,-179.527,6.109,148.959
C04521=1168.786,54.181,-49.270,-179.524,6.111,148.958
C04522=1168.780,54.449,-49.287,-179.521,6.112,148.958
C04523=1168.776,54.718,-49.305,-179.518,6.113,148.957
C04524=1168.770,54.967,-49.321,-179.516,6.114,148.957
C04525=1168.765,55.217,-49.337,-179.513,6.115,148.956
C04526=1168.760,55.466,-49.353,-179.511,6.116,148.956
C04527=1168.755,55.715,-49.369,-179.508,6.117,148.955
C04528=1168.751,55.965,-49.385,-179.505,6.118,148.955
C04529=1168.745,56.214,-49.401,-179.503,6.119,148.954
C04530=1168.741,56.464,-49.418,-179.500,6.120,148.954
C04531=1168.735,56.713,-49.433,-179.497,6.121,148.953
C04532=1168.731,56.963,-49.450,-179.495,6.122,148.953
C04533=1168.725,57.212,-49.466,-179.492,6.123,148.952
C04534=1168.721,57.462,-49.482,-179.490,6.124,148.951
C04535=1168.716,57.711,-49.498,-179.487,6.125,148.951
C04536=1168.711,57.960,-49.514,-179.485,6.126,148.950
C04537=1168.706,58.210,-49.530,-179.482,6.127,148.950
C04538=1168.701,58.459,-49.547,-179.479,6.128,148.949
C04539=1168.695,58.709,-49.563,-179.477,6.129,148.949
C04540=1168.691,58.958,-49.580,-179.474,6.130,148.948
C04541=1168.686,59.207,-49.596,-179.471,6.131,148.947
C04542=1168.681,59.457,-49.612,-179.469,6.132,148.947
C04543=1168.676,59.706,-49.628,-179.466,6.133,148.946
C04544=1168.671,59.956,-49.644,-179.464,6.134,148.946
C04545=1168.666,60.205,-49.660,-179.460,6.135,148.945
C04546=1168.661,60.455,-49.677,-179.458,6.136,148.945
C04547=1168.656,60.704,-49.693,-179.456,6.137,148.944
C04548=1168.651,60.953,-49.709,-179.453,6.138,148.944
C04549=1168.645,61.203,-49.725,-179.450,6.139,148.943
C04550=1168.641,61.453,-49.742,-179.448,6.141,148.943
C04551=1168.636,61.701,-49.758,-179.445,6.141,148.942
C04552=1168.631,61.951,-49.774,-179.443,6.142,148.941
C04553=1168.626,62.200,-49.791,-179.440,6.143,148.941
C04554=1168.621,62.450,-49.807,-179.437,6.144,148.940
C04555=1168.616,62.699,-49.824,-179.434,6.145,148.940
C04556=1168.611,62.949,-49.840,-179.432,6.146,148.939
C04557=1168.606,63.198,-49.857,-179.429,6.147,148.939
C04558=1168.601,63.447,-49.873,-179.427,6.149,148.938
C04559=1168.596,63.697,-49.889,-179.424,6.149,148.938
C04560=1168.591,63.946,-49.905,-179.421,6.151,148.937
C04561=1168.586,64.196,-49.923,-179.419,6.151,148.936
C04562=1168.582,64.445,-49.939,-179.416,6.153,148.936
C04563=1168.577,64.694,-49.956,-179.414,6.154,148.936
C04564=1168.572,64.944,-49.972,-179.411,6.154,148.935
C04565=1168.566,65.193,-49.989,-179.408,6.156,148.934
C04566=1168.561,65.443,-50.005,-179.406,6.156,148.934
C04567=1168.557,65.692,-50.022,-179.403,6.158,148.933
C04568=1168.552,65.941,-50.038,-179.400,6.159,148.933
C04569=1168.546,66.192,-50.055,-179.398,6.160,148.932
C04570=1168.541,66.440,-50.071,-179.395,6.161,148.932
C04571=1168.537,66.690,-50.088,-179.392,6.163,148.931
C04572=1168.532,66.939,-50.104,-179.390,6.163,148.931
C04573=1168.527,67.188,-50.121,-179.388,6.164,148.930
C04574=1168.522,67.438,-50.138,-179.384,6.165,148.929
C04575=1168.518,67.687,-50.155,-179.382,6.166,148.929
C04576=1168.512,67.936,-50.172,-179.379,6.167,148.928
C04577=1168.507,68.186,-50.188,-179.377,6.168,148.928
C04578=1168.503,68.436,-50.204,-179.374,6.170,148.927
C04579=1168.497,68.685,-50.220,-179.371,6.171,148.927
C04580=1168.492,68.935,-50.238,-179.369,6.172,148.926
C04581=1168.488,69.184,-50.254,-179.366,6.173,148.926
C04582=1168.483,69.433,-50.271,-179.363,6.174,148.925
C04583=1168.477,69.683,-50.288,-179.361,6.175,148.925
C04584=1168.473,69.932,-50.305,-179.359,6.176,148.924
C04585=1168.467,70.181,-50.321,-179.355,6.177,148.924
C04586=1168.463,70.431,-50.338,-179.353,6.178,148.923
C04587=1168.458,70.680,-50.355,-179.350,6.179,148.922
C04588=1168.453,70.930,-50.372,-179.348,6.180,148.922
C04589=1168.448,71.179,-50.388,-179.345,6.182,148.922
C04590=1168.443,71.429,-50.406,-179.342,6.182,148.921
C04591=1168.438,71.678,-50.422,-179.340,6.184,148.921
C04592=1168.433,71.927,-50.439,-179.337,6.185,148.920
C04593=1168.428,72.176,-50.457,-179.334,6.186,148.919
C04594=1168.424,72.426,-50.473,-179.332,6.187,148.919
C04595=1168.418,72.675,-50.491,-179.329,6.189,148.918
C04596=1168.413,72.924,-50.507,-179.327,6.189,148.918
C04597=1168.408,73.174,-50.524,-179.324,6.191,148.917
C04598=1168.404,73.423,-50.541,-179.321,6.192,148.917
C04599=1168.399,73.673,-50.557,-179.318,6.193,148.916
C04600=1168.393,73.922,-50.574,-179.316,6.194,148.916
C04601=1168.389,74.171,-50.591,-179.313,6.195,148.915
C04602=1168.384,74.421,-50.609,-179.311,6.196,148.915
C04603=1168.380,74.670,-50.626,-179.308,6.197,148.914
C04604=1168.374,74.919,-50.643,-179.305,6.198,148.914
C04605=1168.369,75.169,-50.659,-179.303,6.200,148.913
C04606=1168.364,75.418,-50.677,-179.300,6.200,148.912
C04607=1168.360,75.667,-50.694,-179.297,6.202,148.912
C04608=1168.355,75.917,-50.711,-179.295,6.203,148.911
C04609=1168.350,76.166,-50.727,-179.292,6.204,148.911
C04610=1168.344,76.416,-50.745,-179.289,6.205,148.910
C04611=1168.339,76.666,-50.762,-179.287,6.207,148.910
C04612=1168.335,76.914,-50.779,-179.284,6.207,148.909
C04613=1168.330,77.164,-50.797,-179.281,6.209,148.909
C04614=1168.325,77.413,-50.813,-179.279,6.210,148.908
C04615=1168.320,77.662,-50.831,-179.276,6.211,148.908
C04616=1168.315,77.912,-50.848,-179.274,6.212,148.907
C04617=1168.310,78.161,-50.865,-179.271,6.214,148.907
C04618=1168.305,78.411,-50.882,-179.268,6.214,148.906
C04619=1168.301,78.660,-50.900,-179.266,6.216,148.906
C04620=1168.295,78.909,-50.916,-179.263,6.216,148.905
C04621=1168.290,79.159,-50.933,-179.260,6.218,148.905
C04622=1168.285,79.408,-50.951,-179.258,6.219,148.904
C04623=1168.280,79.658,-50.968,-179.255,6.220,148.904
C04624=1168.276,79.926,-50.986,-179.252,6.221,148.903
C04625=1168.270,80.194,-51.005,-179.250,6.222,148.903
C04626=1168.264,80.463,-51.024,-179.246,6.224,148.902
C04627=1168.260,80.731,-51.042,-179.244,6.225,148.901
C04628=1168.255,80.980,-51.060,-179.241,6.226,148.901
C04629=1168.250,81.230,-51.077,-179.238,6.228,148.900
C04630=1168.245,81.479,-51.094,-179.236,6.228,148.900
C04631=1168.240,81.728,-51.112,-179.233,6.230,148.899
C04632=1168.234,81.978,-51.129,-179.231,6.231,148.899
C04633=1168.230,82.227,-51.147,-179.228,6.232,148.898
C04634=1168.225,82.477,-51.164,-179.225,6.233,148.898
C04635=1168.220,82.726,-51.182,-179.222,6.234,148.897
C04636=1168.215,82.976,-51.199,-179.219,6.236,148.897
C04637=1168.211,83.224,-51.216,-179.217,6.237,148.896
C04638=1168.206,83.474,-51.234,-179.214,6.238,148.896
C04639=1168.201,83.723,-51.252,-179.212,6.239,148.895
C04640=1168.195,83.973,-51.269,-179.209,6.240,148.895
C04641=1168.191,84.221,-51.286,-179.207,6.241,148.894
C04642=1168.185,84.471,-51.303,-179.204,6.243,148.894
C04643=1168.181,84.720,-51.321,-179.201,6.244,148.893
C04644=1168.176,84.969,-51.339,-179.199,6.245,148.893
C04645=1168.171,85.219,-51.356,-179.196,6.247,148.892
C04646=1168.166,85.468,-51.374,-179.193,6.248,148.892
C04647=1168.161,85.718,-51.391,-179.190,6.249,148.891
C04648=1168.156,85.967,-51.409,-179.188,6.250,148.891
C04649=1168.151,86.216,-51.427,-179.185,6.251,148.890
C04650=1168.147,86.466,-51.444,-179.183,6.252,148.890
C04651=1168.142,86.715,-51.462,-179.180,6.254,148.889
C04652=1168.137,86.965,-51.479,-179.177,6.255,148.889
C04653=1168.132,87.214,-51.497,-179.174,6.256,148.888
C04654=1168.127,87.463,-51.515,-179.172,6.258,148.888
C04655=1168.122,87.713,-51.532,-179.170,6.258,148.887
C04656=1168.117,87.962,-51.549,-179.166,6.260,148.886
C04657=1168.112,88.211,-51.567,-179.164,6.261,148.886
C04658=1168.108,88.460,-51.585,-179.161,6.262,148.886
C04659=1168.102,88.710,-51.603,-179.158,6.264,148.885
C04660=1168.097,88.959,-51.621,-179.156,6.265,148.885
C04661=1168.093,89.208,-51.639,-179.153,6.266,148.884
C04662=1168.088,89.457,-51.657,-179.151,6.267,148.884
C04663=1168.082,89.707,-51.674,-179.148,6.269,148.883
C04664=1168.078,89.956,-51.691,-179.145,6.270,148.882
C04665=1168.073,90.205,-51.709,-179.143,6.271,148.882
C04666=1168.068,90.454,-51.727,-179.140,6.273,148.882
C04667=1168.064,90.705,-51.745,-179.137,6.273,148.881
C04668=1168.059,90.954,-51.763,-179.135,6.275,148.881
C04669=1168.054,91.203,-51.781,-179.132,6.276,148.880
C04670=1168.049,91.452,-51.799,-179.129,6.277,148.879
C04671=1168.044,91.702,-51.817,-179.127,6.279,148.879
C04672=1168.039,91.951,-51.835,-179.124,6.279,148.878
C04673=1168.034,92.201,-51.852,-179.121,6.281,148.878
C04674=1168.029,92.450,-51.870,-179.118,6.283,148.878
C04675=1168.024,92.699,-51.888,-179.116,6.283,148.877
C04676=1168.019,92.948,-51.906,-179.113,6.285,148.877
C04677=1168.014,93.197,-51.924,-179.110,6.287,148.876
C04678=1168.009,93.446,-51.942,-179.108,6.287,148.875
C04679=1168.005,93.696,-51.960,-179.105,6.289,148.875
C04680=1168.000,93.946,-51.978,-179.103,6.290,148.875
C04681=1167.995,94.195,-51.996,-179.100,6.291,148.874
C04682=1167.990,94.444,-52.014,-179.097,6.293,148.874
C04683=1167.985,94.693,-52.032,-179.095,6.294,148.873
C04684=1167.981,94.942,-52.050,-179.092,6.295,148.872
C04685=1167.976,95.191,-52.068,-179.089,6.297,148.872
C04686=1167.971,95.441,-52.086,-179.087,6.298,148.872
C04687=1167.966,95.690,-52.104,-179.084,6.299,148.871
C04688=1167.962,95.940,-52.122,-179.081,6.300,148.871
C04689=1167.957,96.189,-52.140,-179.079,6.302,148.870
C04690=1167.952,96.438,-52.158,-179.076,6.303,148.870
C04691=1167.946,96.687,-52.177,-179.073,6.304,148.869
C04692=1167.941,96.937,-52.195,-179.071,6.305,148.869
C04693=1167.937,97.187,-52.213,-179.067,6.307,148.868
C04694=1167.932,97.436,-52.231,-179.065,6.308,148.868
C04695=1167.927,97.685,-52.249,-179.063,6.309,148.867
C04696=1167.922,97.934,-52.267,-179.059,6.311,148.867
C04697=1167.917,98.183,-52.285,-179.057,6.312,148.866
C04698=1167.912,98.432,-52.303,-179.055,6.313,148.866
C04699=1167.907,98.683,-52.322,-179.051,6.315,148.865
C04700=1167.902,98.932,-52.340,-179.049,6.316,148.865
C04701=1167.898,99.180,-52.359,-179.046,6.317,148.864
C04702=1167.893,99.429,-52.377,-179.043,6.319,148.864
C04703=1167.888,99.679,-52.395,-179.041,6.320,148.863
C04704=1167.884,99.929,-52.413,-179.038,6.321,148.863
C04705=1167.878,100.178,-52.432,-179.035,6.323,148.862
C04706=1167.873,100.427,-52.450,-179.033,6.324,148.862
C04707=1167.868,100.676,-52.468,-179.030,6.325,148.861
C04708=1167.864,100.926,-52.487,-179.027,6.327,148.861
C04709=1167.859,101.175,-52.505,-179.025,6.328,148.860
C04710=1167.854,101.424,-52.523,-179.022,6.329,148.860
C04711=1167.849,101.673,-52.542,-179.020,6.331,148.859
C04712=1167.845,101.923,-52.560,-179.017,6.331,148.859
C04713=1167.840,102.172,-52.578,-179.014,6.333,148.858
C04714=1167.834,102.421,-52.597,-179.012,6.335,148.858
C04715=1167.829,102.670,-52.616,-179.009,6.335,148.857
C04716=1167.825,102.920,-52.634,-179.006,6.337,148.857
C04717=1167.820,103.169,-52.652,-179.003,6.339,148.857
C04718=1167.815,103.418,-52.671,-179.001,6.339,148.856
C04719=1167.811,103.668,-52.690,-178.998,6.341,148.855
C04720=1167.806,103.917,-52.708,-178.995,6.343,148.855
C04721=1167.800,104.166,-52.727,-178.993,6.344,148.855
C04722=1167.796,104.416,-52.745,-178.990,6.345,148.854
C04723=1167.791,104.665,-52.763,-178.987,6.347,148.854
C04724=1167.786,104.914,-52.782,-178.985,6.348,148.853
C04725=1167.781,105.163,-52.800,-178.982,6.349,148.853
C04726=1167.776,105.413,-52.819,-178.979,6.351,148.852
C04727=1167.771,105.662,-52.838,-178.977,6.352,148.852
C04728=1167.766,105.930,-52.857,-178.973,6.354,148.851
C04729=1167.761,106.199,-52.878,-178.971,6.355,148.851
C04730=1167.756,106.467,-52.898,-178.968,6.356,148.850
C04731=1167.750,106.735,-52.918,-178.965,6.358,148.850
C04732=1167.746,106.985,-52.937,-178.963,6.360,148.849
C04733=1167.741,107.234,-52.956,-178.959,6.361,148.849
C04734=1167.736,107.483,-52.974,-178.957,6.362,148.848
C04735=1167.732,107.733,-52.993,-178.955,6.363,148.848
C04736=1167.726,107.981,-53.012,-178.952,6.365,148.847
C04737=1167.721,108.231,-53.030,-178.949,6.367,148.847
C04738=1167.717,108.480,-53.050,-178.947,6.367,148.846
C04739=1167.712,108.729,-53.068,-178.944,6.369,148.846
C04740=1167.707,108.978,-53.086,-178.941,6.371,148.845
C04741=1167.702,109.228,-53.105,-178.938,6.371,148.845
C04742=1167.698,109.477,-53.124,-178.936,6.373,148.844
C04743=1167.692,109.727,-53.143,-178.933,6.375,148.844
C04744=1167.688,109.975,-53.162,-178.930,6.376,148.843
C04745=1167.683,110.225,-53.181,-178.928,6.377,148.843
C04746=1167.678,110.474,-53.199,-178.925,6.379,148.843
C04747=1167.673,110.723,-53.218,-178.922,6.381,148.842
C04748=1167.669,110.973,-53.237,-178.919,6.382,148.842
C04749=1167.663,111.222,-53.256,-178.917,6.383,148.841
C04750=1167.659,111.471,-53.275,-178.914,6.385,148.841
C04751=1167.654,111.720,-53.294,-178.912,6.386,148.840
C04752=1167.650,111.970,-53.313,-178.908,6.388,148.840
C04753=1167.644,112.219,-53.332,-178.906,6.389,148.839
C04754=1167.639,112.468,-53.350,-178.903,6.390,148.839
C04755=1167.635,112.717,-53.370,-178.901,6.392,148.838
C04756=1167.630,112.966,-53.388,-178.898,6.393,148.838
C04757=1167.625,113.215,-53.408,-178.895,6.394,148.837
C04758=1167.620,113.465,-53.427,-178.893,6.396,148.837
C04759=1167.616,113.714,-53.446,-178.890,6.398,148.837
C04760=1167.610,113.963,-53.465,-178.887,6.399,148.836
C04761=1167.606,114.213,-53.483,-178.885,6.400,148.836
C04762=1167.601,114.462,-53.503,-178.882,6.402,148.835
C04763=1167.596,114.711,-53.522,-178.879,6.403,148.835
C04764=1167.591,114.960,-53.541,-178.876,6.405,148.834
C04765=1167.586,115.209,-53.561,-178.874,6.406,148.834
C04766=1167.582,115.459,-53.579,-178.871,6.407,148.833
C04767=1167.577,115.708,-53.598,-178.869,6.409,148.833
C04768=1167.571,115.957,-53.618,-178.866,6.411,148.833
C04769=1167.567,116.206,-53.637,-178.863,6.412,148.832
C04770=1167.562,116.455,-53.656,-178.860,6.413,148.832
C04771=1167.557,116.705,-53.676,-178.858,6.415,148.831
C04772=1167.553,116.953,-53.694,-178.855,6.417,148.831
C04773=1167.548,117.204,-53.713,-178.852,6.418,148.830
C04774=1167.542,117.452,-53.732,-178.850,6.419,148.830
C04775=1167.538,117.702,-53.752,-178.847,6.421,148.829
C04776=1167.533,117.951,-53.771,-178.844,6.422,148.829
C04777=1167.528,118.200,-53.790,-178.842,6.424,148.828
C04778=1167.524,118.450,-53.810,-178.838,6.425,148.828
C04779=1167.519,118.698,-53.829,-178.836,6.426,148.827
C04780=1167.514,118.948,-53.848,-178.834,6.428,148.827
C04781=1167.509,119.197,-53.868,-178.831,6.430,148.827
C04782=1167.505,119.446,-53.887,-178.828,6.431,148.826
C04783=1167.499,119.695,-53.906,-178.825,6.433,148.826
C04784=1167.495,119.944,-53.926,-178.823,6.434,148.825
C04785=1167.490,120.194,-53.945,-178.820,6.435,148.825
C04786=1167.485,120.442,-53.964,-178.817,6.437,148.824
C04787=1167.481,120.692,-53.984,-178.814,6.438,148.824
C04788=1167.475,120.941,-54.003,-178.811,6.440,148.823
C04789=1167.471,121.190,-54.023,-178.809,6.441,148.823
C04790=1167.466,121.440,-54.042,-178.807,6.443,148.823
C04791=1167.461,121.689,-54.061,-178.804,6.445,148.822
C04792=1167.456,121.938,-54.081,-178.801,6.446,148.822
C04793=1167.452,122.188,-54.100,-178.798,6.448,148.821
C04794=1167.447,122.436,-54.120,-178.795,6.449,148.821
C04795=1167.442,122.686,-54.140,-178.793,6.450,148.820
C04796=1167.437,122.934,-54.159,-178.790,6.452,148.820
C04797=1167.433,123.184,-54.178,-178.787,6.453,148.819
C04798=1167.428,123.433,-54.198,-178.785,6.455,148.819
C04799=1167.423,123.682,-54.217,-178.782,6.457,148.819
C04800=1167.418,123.932,-54.237,-178.780,6.458,148.818
C04801=1167.413,124.181,-54.257,-178.777,6.459,148.818
C04802=1167.408,124.429,-54.277,-178.774,6.461,148.817
C04803=1167.403,124.679,-54.296,-178.771,6.463,148.817
C04804=1167.398,124.929,-54.316,-178.768,6.464,148.816
C04805=1167.394,125.178,-54.335,-178.766,6.466,148.816
C04806=1167.389,125.426,-54.355,-178.764,6.467,148.815
C04807=1167.385,125.676,-54.375,-178.761,6.469,148.815
C04808=1167.380,125.925,-54.394,-178.758,6.470,148.815
C04809=1167.375,126.174,-54.414,-178.755,6.472,148.814
C04810=1167.370,126.423,-54.434,-178.752,6.474,148.814
C04811=1167.365,126.673,-54.454,-178.750,6.475,148.813
C04812=1167.361,126.922,-54.473,-178.747,6.477,148.813
C04813=1167.356,127.170,-54.493,-178.745,6.478,148.812
C04814=1167.351,127.420,-54.513,-178.742,6.480,148.812
C04815=1167.346,127.670,-54.533,-178.739,6.481,148.811
C04816=1167.341,127.918,-54.553,-178.736,6.483,148.811
C04817=1167.336,128.167,-54.572,-178.733,6.484,148.811
C04818=1167.332,128.417,-54.592,-178.731,6.486,148.810
C04819=1167.327,128.666,-54.612,-178.728,6.488,148.810
C04820=1167.322,128.915,-54.632,-178.726,6.489,148.809
C04821=1167.317,129.164,-54.651,-178.723,6.490,148.809
C04822=1167.313,129.413,-54.672,-178.720,6.492,148.808
C04823=1167.308,129.663,-54.691,-178.717,6.494,148.808
C04824=1167.304,129.912,-54.712,-178.715,6.495,148.808
C04825=1167.298,130.161,-54.731,-178.712,6.497,148.807
C04826=1167.294,130.410,-54.751,-178.709,6.499,148.807
C04827=1167.289,130.659,-54.771,-178.706,6.501,148.807
C04828=1167.285,130.908,-54.791,-178.704,6.501,148.806
C04829=1167.279,131.157,-54.811,-178.701,6.503,148.805
C04830=1167.275,131.406,-54.831,-178.698,6.505,148.805
C04831=1167.269,131.656,-54.851,-178.696,6.506,148.805
C04832=1167.264,131.925,-54.872,-178.693,6.508,148.804
C04833=1167.260,132.193,-54.894,-178.690,6.509,148.804
C04834=1167.254,132.462,-54.916,-178.687,6.511,148.803
C04835=1167.249,132.730,-54.937,-178.684,6.514,148.803
C04836=1167.245,132.979,-54.957,-178.682,6.515,148.803
C04837=1167.240,133.228,-54.978,-178.679,6.516,148.802
C04838=1167.235,133.478,-54.998,-178.676,6.518,148.802
C04839=1167.230,133.726,-55.018,-178.673,6.519,148.801
C04840=1167.225,133.976,-55.038,-178.670,6.521,148.801
C04841=1167.221,134.225,-55.058,-178.668,6.523,148.800
C04842=1167.216,134.474,-55.078,-178.665,6.525,148.800
C04843=1167.211,134.724,-55.099,-178.662,6.526,148.800
C04844=1167.206,134.972,-55.119,-178.660,6.528,148.799
C04845=1167.202,135.222,-55.139,-178.657,6.530,148.799
C04846=1167.197,135.471,-55.159,-178.655,6.531,148.798
C04847=1167.192,135.719,-55.179,-178.652,6.532,148.798
C04848=1167.187,135.969,-55.200,-178.649,6.534,148.797
C04849=1167.182,136.218,-55.220,-178.646,6.536,148.797
C04850=1167.178,136.467,-55.240,-178.644,6.537,148.797
C04851=1167.173,136.716,-55.260,-178.641,6.539,148.796
C04852=1167.168,136.966,-55.281,-178.638,6.541,148.796
C04853=1167.163,137.215,-55.301,-178.635,6.543,148.795
C04854=1167.159,137.464,-55.321,-178.633,6.544,148.795
C04855=1167.154,137.713,-55.342,-178.630,6.546,148.795
C04856=1167.149,137.963,-55.362,-178.627,6.547,148.794
C04857=1167.145,138.212,-55.382,-178.624,6.549,148.794
C04858=1167.140,138.460,-55.402,-178.621,6.551,148.793
C04859=1167.134,138.709,-55.423,-178.619,6.553,148.793
C04860=1167.130,138.958,-55.444,-178.617,6.554,148.792
C04861=1167.125,139.208,-55.463,-178.614,6.555,148.792
C04862=1167.120,139.457,-55.484,-178.611,6.557,148.792
C04863=1167.116,139.706,-55.505,-178.608,6.559,148.791
C04864=1167.111,139.955,-55.525,-178.606,6.560,148.791
C04865=1167.106,140.204,-55.546,-178.603,6.562,148.791
C04866=1167.101,140.453,-55.566,-178.600,6.564,148.790
C04867=1167.097,140.702,-55.587,-178.598,6.566,148.790
C04868=1167.092,140.951,-55.608,-178.594,6.567,148.789
C04869=1167.087,141.200,-55.628,-178.592,6.569,148.789
C04870=1167.083,141.450,-55.648,-178.589,6.571,148.788
C04871=1167.078,141.699,-55.669,-178.586,6.572,148.788
C04872=1167.073,141.948,-55.689,-178.584,6.574,148.788
C04873=1167.068,142.197,-55.710,-178.581,6.576,148.787
C04874=1167.063,142.446,-55.730,-178.578,6.578,148.787
C04875=1167.059,142.695,-55.751,-178.576,6.579,148.786
C04876=1167.054,142.944,-55.772,-178.573,6.581,148.786
C04877=1167.049,143.193,-55.792,-178.570,6.583,148.786
C04878=1167.044,143.442,-55.813,-178.567,6.584,148.785
C04879=1167.040,143.691,-55.834,-178.565,6.586,148.785
C04880=1167.035,143.941,-55.854,-178.562,6.588,148.785
C04881=1167.030,144.190,-55.875,-178.559,6.590,148.784
C04882=1167.026,144.439,-55.897,-178.557,6.591,148.784
C04883=1167.021,144.688,-55.917,-178.555,6.592,148.783
C04884=1167.016,144.937,-55.938,-178.551,6.594,148.783
C04885=1167.012,145.186,-55.959,-178.549,6.595,148.782
C04886=1167.007,145.435,-55.980,-178.546,6.597,148.782
C04887=1167.002,145.684,-56.000,-178.543,6.599,148.782
C04888=1166.997,145.934,-56.021,-178.541,6.601,148.781
C04889=1166.993,146.183,-56.041,-178.538,6.602,148.781
C04890=1166.987,146.432,-56.062,-178.535,6.604,148.780
C04891=1166.983,146.680,-56.083,-178.532,6.606,148.780
C04892=1166.978,146.929,-56.104,-178.530,6.608,148.780
C04893=1166.974,147.178,-56.125,-178.527,6.609,148.779
C04894=1166.969,147.428,-56.146,-178.524,6.611,148.779
C04895=1166.965,147.677,-56.166,-178.522,6.613,148.779
C04896=1166.960,147.926,-56.188,-178.519,6.615,148.778
C04897=1166.955,148.175,-56.209,-178.516,6.616,148.778
C04898=1166.950,148.424,-56.229,-178.514,6.618,148.777
C04899=1166.945,148.673,-56.250,-178.511,6.620,148.777
C04900=1166.941,148.922,-56.271,-178.508,6.622,148.777
C04901=1166.936,149.171,-56.292,-178.505,6.623,148.776
C04902=1166.931,149.421,-56.314,-178.503,6.625,148.776
C04903=1166.927,149.670,-56.334,-178.500,6.627,148.775
C04904=1166.922,149.918,-56.356,-178.497,6.629,148.775
C04905=1166.917,150.168,-56.377,-178.495,6.630,148.775
C04906=1166.912,150.417,-56.397,-178.492,6.632,148.774
C04907=1166.907,150.665,-56.419,-178.489,6.634,148.774
C04908=1166.903,150.915,-56.440,-178.486,6.636,148.774
C04909=1166.898,151.164,-56.461,-178.483,6.638,148.773
C04910=1166.894,151.413,-56.482,-178.481,6.640,148.773
C04911=1166.888,151.662,-56.503,-178.478,6.642,148.772
C04912=1166.884,151.911,-56.524,-178.475,6.643,148.772
C04913=1166.879,152.160,-56.545,-178.473,6.645,148.772
C04914=1166.874,152.410,-56.567,-178.470,6.647,148.771
C04915=1166.870,152.658,-56.588,-178.467,6.649,148.771
C04916=1166.865,152.907,-56.609,-178.464,6.650,148.771
C04917=1166.860,153.156,-56.630,-178.462,6.652,148.770
C04918=1166.856,153.406,-56.652,-178.459,6.654,148.770
C04919=1166.851,153.655,-56.673,-178.456,6.656,148.769
C04920=1166.846,153.903,-56.694,-178.454,6.657,148.769
C04921=1166.842,154.152,-56.715,-178.451,6.659,148.769
C04922=1166.836,154.401,-56.736,-178.448,6.661,148.768
C04923=1166.832,154.651,-56.758,-178.446,6.663,148.768
C04924=1166.828,154.900,-56.779,-178.443,6.664,148.768
C04925=1166.823,155.148,-56.800,-178.440,6.666,148.767
C04926=1166.818,155.398,-56.821,-178.438,6.668,148.767
C04927=1166.813,155.647,-56.843,-178.435,6.670,148.766
C04928=1166.808,155.896,-56.864,-178.432,6.671,148.766
C04929=1166.804,156.144,-56.886,-178.429,6.673,148.766
C04930=1166.799,156.394,-56.907,-178.427,6.675,148.765
C04931=1166.795,156.643,-56.929,-178.423,6.677,148.765
C04932=1166.790,156.892,-56.950,-178.421,6.679,148.765
C04933=1166.785,157.141,-56.971,-178.418,6.681,148.764
C04934=1166.780,157.390,-56.993,-178.415,6.683,148.764
C04935=1166.775,157.639,-57.015,-178.413,6.684,148.763
C04936=1166.771,157.908,-57.038,-178.410,6.686,148.763
C04937=1166.765,158.177,-57.061,-178.407,6.688,148.763
C04938=1166.760,158.446,-57.084,-178.404,6.690,148.762
C04939=1166.755,158.715,-57.108,-178.401,6.692,148.762
C04940=1166.750,158.964,-57.129,-178.399,6.694,148.762
C04941=1166.746,159.213,-57.150,-178.396,6.696,148.761
C04942=1166.742,159.462,-57.172,-178.393,6.697,148.761
C04943=1166.737,159.711,-57.194,-178.391,6.699,148.760
C04944=1166.732,159.960,-57.215,-178.388,6.701,148.760
C04945=1166.727,160.209,-57.237,-178.385,6.703,148.760
C04946=1166.723,160.458,-57.258,-178.382,6.705,148.759
C04947=1166.718,160.707,-57.280,-178.379,6.707,148.759
C04948=1166.713,160.956,-57.302,-178.377,6.709,148.759
C04949=1166.708,161.205,-57.323,-178.374,6.710,148.758
C04950=1166.704,161.455,-57.345,-178.371,6.712,148.758
C04951=1166.699,161.703,-57.367,-178.369,6.714,148.758
C04952=1166.694,161.952,-57.388,-178.366,6.716,148.757
C04953=1166.690,162.201,-57.411,-178.364,6.718,148.757
C04954=1166.685,162.450,-57.432,-178.361,6.720,148.757
C04955=1166.680,162.700,-57.454,-178.358,6.722,148.756
C04956=1166.676,162.948,-57.475,-178.355,6.724,148.756
C04957=1166.671,163.198,-57.497,-178.352,6.726,148.755
C04958=1166.666,163.446,-57.519,-178.350,6.727,148.755
C04959=1166.662,163.695,-57.541,-178.347,6.729,148.755
C04960=1166.657,163.944,-57.563,-178.344,6.731,148.754
C04961=1166.652,164.193,-57.584,-178.341,6.733,148.754
C04962=1166.648,164.442,-57.606,-178.339,6.734,148.754
C04963=1166.643,164.691,-57.629,-178.336,6.736,148.753
C04964=1166.638,164.941,-57.651,-178.333,6.739,148.753
C04965=1166.633,165.189,-57.672,-178.331,6.741,148.753
C04966=1166.629,165.439,-57.694,-178.328,6.743,148.752
C04967=1166.624,165.687,-57.716,-178.325,6.744,148.752
C04968=1166.619,165.936,-57.738,-178.322,6.746,148.752
C04969=1166.615,166.185,-57.760,-178.320,6.748,148.751
C04970=1166.610,166.434,-57.782,-178.317,6.750,148.751
C04971=1166.606,166.683,-57.804,-178.314,6.752,148.751
C04972=1166.600,166.932,-57.826,-178.311,6.754,148.750
C04973=1166.596,167.182,-57.848,-178.308,6.756,148.750
C04974=1166.591,167.430,-57.870,-178.306,6.758,148.750
C04975=1166.587,167.680,-57.892,-178.304,6.759,148.749
C04976=1166.582,167.928,-57.914,-178.301,6.761,148.749
C04977=1166.577,168.177,-57.937,-178.298,6.763,148.749
C04978=1166.573,168.426,-57.958,-178.295,6.766,148.748
C04979=1166.568,168.675,-57.980,-178.292,6.767,148.748
C04980=1166.563,168.924,-58.002,-178.290,6.769,148.747
C04981=1166.558,169.173,-58.025,-178.287,6.771,148.747
C04982=1166.554,169.422,-58.048,-178.285,6.773,148.747
C04983=1166.550,169.671,-58.069,-178.282,6.775,148.747
C04984=1166.545,169.920,-58.091,-178.279,6.776,148.746
C04985=1166.540,170.169,-58.114,-178.276,6.779,148.746
C04986=1166.535,170.418,-58.136,-178.273,6.781,148.745
C04987=1166.531,170.666,-58.158,-178.271,6.783,148.745
C04988=1166.527,170.916,-58.180,-178.268,6.784,148.745
C04989=1166.521,171.165,-58.202,-178.265,6.786,148.744
C04990=1166.517,171.414,-58.224,-178.263,6.788,148.744
C04991=1166.513,171.663,-58.247,-178.260,6.791,148.744
C04992=1166.507,171.912,-58.269,-178.257,6.792,148.744
C04993=1166.503,172.161,-58.291,-178.254,6.794,148.743
C04994=1166.498,172.409,-58.314,-178.252,6.796,148.743
C04995=1166.493,172.659,-58.337,-178.249,6.798,148.742
C04996=1166.489,172.908,-58.359,-178.246,6.801,148.742
C04997=1166.485,173.156,-58.381,-178.244,6.802,148.742
C04998=1166.480,173.406,-58.404,-178.241,6.804,148.742
C04999=1166.475,173.654,-58.425,-178.238,6.806,148.741
C05000=1166.471,173.903,-58.448,-178.235,6.808,148.741
C05001=1166.466,174.153,-58.471,-178.233,6.809,148.740
C05002=1166.461,174.401,-58.493,-178.230,6.812,148.740
C05003=1166.456,174.651,-58.516,-178.227,6.814,148.740
C05004=1166.452,174.899,-58.538,-178.225,6.816,148.740
C05005=1166.447,175.148,-58.560,-178.222,6.818,148.739
C05006=1166.442,175.398,-58.583,-178.219,6.819,148.739
C05007=1166.438,175.646,-58.605,-178.216,6.822,148.739
C05008=1166.433,175.895,-58.628,-178.213,6.824,148.738
C05009=1166.429,176.144,-58.651,-178.211,6.826,148.738
C05010=1166.424,176.394,-58.673,-178.208,6.828,148.738
C05011=1166.419,176.642,-58.696,-178.206,6.829,148.737
C05012=1166.415,176.890,-58.718,-178.202,6.832,148.737
C05013=1166.410,177.140,-58.741,-178.200,6.834,148.737
C05014=1166.406,177.388,-58.763,-178.198,6.836,148.736
C05015=1166.401,177.638,-58.786,-178.195,6.838,148.736
C05016=1166.397,177.886,-58.809,-178.192,6.840,148.736
C05017=1166.391,178.135,-58.831,-178.189,6.842,148.735
C05018=1166.387,178.384,-58.854,-178.186,6.844,148.735
C05019=1166.382,178.633,-58.877,-178.184,6.846,148.735
C05020=1166.378,178.882,-58.899,-178.181,6.848,148.735
C05021=1166.373,179.131,-58.922,-178.178,6.850,148.734
C05022=1166.368,179.380,-58.946,-178.175,6.852,148.734
C05023=1166.364,179.629,-58.968,-178.173,6.854,148.733
C05024=1166.359,179.877,-58.991,-178.171,6.856,148.733
C05025=1166.355,180.126,-59.013,-178.167,6.858,148.733
C05026=1166.350,180.376,-59.036,-178.165,6.860,148.733
C05027=1166.346,180.625,-59.059,-178.162,6.862,148.732
C05028=1166.341,180.874,-59.082,-178.159,6.864,148.732
C05029=1166.335,181.123,-59.105,-178.156,6.867,148.732
C05030=1166.331,181.371,-59.127,-178.154,6.868,148.731
C05031=1166.327,181.620,-59.151,-178.151,6.870,148.731
C05032=1166.323,181.869,-59.173,-178.148,6.872,148.731
C05033=1166.317,182.118,-59.196,-178.146,6.875,148.731
C05034=1166.312,182.367,-59.219,-178.143,6.876,148.730
C05035=1166.308,182.616,-59.242,-178.140,6.878,148.730
C05036=1166.304,182.865,-59.265,-178.138,6.880,148.729
C05037=1166.299,183.114,-59.289,-178.134,6.883,148.729
C05038=1166.294,183.362,-59.311,-178.132,6.885,148.729
C05039=1166.289,183.611,-59.334,-178.129,6.886,148.729
C05040=1166.284,183.881,-59.359,-178.126,6.889,148.728
C05041=1166.280,184.150,-59.384,-178.123,6.891,148.728
C05042=1166.275,184.420,-59.409,-178.120,6.893,148.728
C05043=1166.269,184.690,-59.434,-178.118,6.895,148.727
C05044=1166.265,184.938,-59.457,-178.115,6.897,148.727
C05045=1166.261,185.187,-59.480,-178.112,6.900,148.727
C05046=1166.256,185.436,-59.503,-178.109,6.902,148.726
C05047=1166.251,185.685,-59.527,-178.107,6.903,148.726
C05048=1166.247,185.934,-59.549,-178.104,6.906,148.726
C05049=1166.243,186.183,-59.573,-178.101,6.908,148.726
C05050=1166.237,186.431,-59.596,-178.099,6.910,148.725
C05051=1166.233,186.680,-59.619,-178.096,6.912,148.725
C05052=1166.229,186.929,-59.642,-178.093,6.915,148.725
C05053=1166.224,187.178,-59.665,-178.090,6.916,148.724
C05054=1166.219,187.427,-59.689,-178.088,6.918,148.724
C05055=1166.214,187.676,-59.712,-178.084,6.921,148.724
C05056=1166.210,187.925,-59.735,-178.082,6.923,148.724
C05057=1166.206,188.174,-59.758,-178.080,6.925,148.723
C05058=1166.201,188.423,-59.781,-178.077,6.926,148.723
C05059=1166.196,188.672,-59.805,-178.074,6.929,148.723
C05060=1166.191,188.920,-59.828,-178.071,6.931,148.722
C05061=1166.186,189.170,-59.851,-178.069,6.933,148.722
C05062=1166.182,189.419,-59.875,-178.066,6.935,148.722
C05063=1166.177,189.668,-59.898,-178.063,6.937,148.722
C05064=1166.173,189.916,-59.921,-178.061,6.939,148.721
C05065=1166.169,190.165,-59.945,-178.057,6.942,148.721
C05066=1166.164,190.414,-59.968,-178.055,6.944,148.721
C05067=1166.159,190.663,-59.991,-178.053,6.946,148.720
C05068=1166.155,190.912,-60.015,-178.050,6.947,148.720
C05069=1166.150,191.161,-60.038,-178.047,6.950,148.720
C05070=1166.145,191.409,-60.062,-178.044,6.952,148.720
C05071=1166.141,191.658,-60.086,-178.042,6.954,148.719
C05072=1166.136,191.907,-60.109,-178.038,6.957,148.719
C05073=1166.131,192.156,-60.132,-178.036,6.959,148.719
C05074=1166.127,192.405,-60.156,-178.034,6.960,148.718
C05075=1166.122,192.654,-60.180,-178.030,6.963,148.718
C05076=1166.118,192.903,-60.203,-178.028,6.965,148.718
C05077=1166.113,193.151,-60.227,-178.025,6.967,148.718
C05078=1166.108,193.400,-60.251,-178.022,6.969,148.717
C05079=1166.104,193.649,-60.274,-178.019,6.971,148.717
C05080=1166.099,193.898,-60.297,-178.017,6.973,148.717
C05081=1166.095,194.147,-60.321,-178.014,6.976,148.716
C05082=1166.090,194.396,-60.345,-178.011,6.978,148.716
C05083=1166.086,194.644,-60.369,-178.009,6.980,148.716
C05084=1166.081,194.893,-60.392,-178.006,6.982,148.716
C05085=1166.076,195.142,-60.415,-178.003,6.984,148.715
C05086=1166.072,195.391,-60.440,-178.001,6.986,148.715
C05087=1166.067,195.640,-60.463,-177.998,6.989,148.715
C05088=1166.063,195.888,-60.487,-177.995,6.991,148.715
C05089=1166.058,196.137,-60.510,-177.993,6.993,148.714
C05090=1166.054,196.386,-60.534,-177.990,6.995,148.714
C05091=1166.049,196.635,-60.558,-177.987,6.997,148.714
C05092=1166.045,196.884,-60.582,-177.985,6.999,148.714
C05093=1166.040,197.133,-60.606,-177.982,7.002,148.713
C05094=1166.035,197.382,-60.630,-177.979,7.004,148.713
C05095=1166.031,197.630,-60.654,-177.976,7.007,148.713
C05096=1166.026,197.879,-60.678,-177.973,7.008,148.712
C05097=1166.021,198.128,-60.701,-177.971,7.010,148.712
C05098=1166.017,198.376,-60.725,-177.968,7.013,148.712
C05099=1166.012,198.625,-60.748,-177.965,7.015,148.712
C05100=1166.008,198.874,-60.773,-177.963,7.017,148.712
C05101=1166.003,199.124,-60.797,-177.960,7.019,148.711
C05102=1165.999,199.372,-60.821,-177.957,7.021,148.711
C05103=1165.994,199.621,-60.845,-177.954,7.024,148.711
C05104=1165.990,199.870,-60.868,-177.952,7.026,148.710
C05105=1165.985,200.118,-60.892,-177.949,7.028,148.710
C05106=1165.980,200.367,-60.916,-177.946,7.031,148.710
C05107=1165.975,200.616,-60.940,-177.944,7.032,148.710
C05108=1165.972,200.865,-60.965,-177.941,7.035,148.709
C05109=1165.967,201.114,-60.988,-177.938,7.037,148.709
C05110=1165.963,201.362,-61.012,-177.935,7.039,148.709
C05111=1165.957,201.611,-61.037,-177.933,7.042,148.709
C05112=1165.953,201.860,-61.061,-177.930,7.044,148.708
C05113=1165.949,202.109,-61.085,-177.927,7.045,148.708
C05114=1165.944,202.358,-61.109,-177.925,7.048,148.708
C05115=1165.939,202.606,-61.134,-177.922,7.050,148.708
C05116=1165.935,202.855,-61.158,-177.919,7.053,148.707
C05117=1165.930,203.104,-61.181,-177.916,7.055,148.707
C05118=1165.926,203.353,-61.206,-177.914,7.057,148.707
C05119=1165.921,203.602,-61.230,-177.911,7.060,148.707
C05120=1165.917,203.850,-61.254,-177.908,7.061,148.706
C05121=1165.912,204.099,-61.279,-177.905,7.064,148.706
C05122=1165.907,204.347,-61.303,-177.903,7.066,148.706
C05123=1165.903,204.597,-61.327,-177.900,7.068,148.706
C05124=1165.898,204.846,-61.351,-177.897,7.071,148.705
C05125=1165.894,205.094,-61.375,-177.895,7.073,148.705
C05126=1165.889,205.343,-61.399,-177.892,7.075,148.705
C05127=1165.885,205.592,-61.425,-177.889,7.077,148.705
C05128=1165.881,205.840,-61.449,-177.887,7.079,148.705
C05129=1165.875,206.089,-61.473,-177.884,7.082,148.704
C05130=1165.871,206.338,-61.497,-177.881,7.084,148.704
C05131=1165.867,206.587,-61.522,-177.878,7.087,148.704
C05132=1165.862,206.835,-61.546,-177.876,7.088,148.703
C05133=1165.858,207.084,-61.571,-177.873,7.091,148.703
C05134=1165.853,207.333,-61.596,-177.870,7.093,148.703
C05135=1165.849,207.582,-61.620,-177.868,7.095,148.703
C05136=1165.844,207.830,-61.644,-177.865,7.098,148.703
C05137=1165.840,208.079,-61.669,-177.862,7.100,148.702
C05138=1165.835,208.328,-61.693,-177.859,7.103,148.702
C05139=1165.830,208.577,-61.717,-177.857,7.104,148.702
C05140=1165.825,208.825,-61.742,-177.854,7.107,148.702
C05141=1165.821,209.074,-61.767,-177.851,7.109,148.701
C05142=1165.816,209.323,-61.791,-177.848,7.112,148.701
C05143=1165.812,209.572,-61.815,-177.846,7.114,148.701
C05144=1165.807,209.842,-61.842,-177.843,7.116,148.701
C05145=1165.802,210.113,-61.869,-177.840,7.119,148.700
C05146=1165.798,210.383,-61.896,-177.837,7.121,148.700
C05147=1165.792,210.654,-61.923,-177.834,7.124,148.700
C05148=1165.787,210.902,-61.948,-177.832,7.126,148.700
C05149=1165.784,211.151,-61.972,-177.828,7.128,148.699
C05150=1165.778,211.400,-61.997,-177.826,7.131,148.699
C05151=1165.774,211.649,-62.021,-177.823,7.133,148.699
C05152=1165.769,211.898,-62.046,-177.821,7.135,148.699
C05153=1165.765,212.146,-62.071,-177.818,7.138,148.698
C05154=1165.761,212.395,-62.096,-177.815,7.140,148.698
C05155=1165.756,212.644,-62.120,-177.812,7.143,148.698
C05156=1165.751,212.892,-62.144,-177.810,7.145,148.698
C05157=1165.747,213.141,-62.170,-177.807,7.147,148.698
C05158=1165.742,213.390,-62.195,-177.804,7.149,148.698
C05159=1165.738,213.639,-62.219,-177.801,7.152,148.697
C05160=1165.733,213.887,-62.245,-177.799,7.154,148.697
C05161=1165.729,214.137,-62.270,-177.796,7.157,148.697
C05162=1165.724,214.385,-62.294,-177.794,7.159,148.697
C05163=1165.720,214.633,-62.319,-177.790,7.161,148.696
C05164=1165.715,214.882,-62.344,-177.788,7.164,148.696
C05165=1165.711,215.131,-62.368,-177.785,7.166,148.696
C05166=1165.706,215.380,-62.394,-177.783,7.168,148.696
C05167=1165.701,215.628,-62.419,-177.779,7.171,148.695
C05168=1165.698,215.877,-62.444,-177.777,7.173,148.695
C05169=1165.693,216.126,-62.468,-177.775,7.175,148.695
C05170=1165.688,216.375,-62.493,-177.772,7.178,148.695
C05171=1165.683,216.623,-62.519,-177.769,7.180,148.695
C05172=1165.680,216.872,-62.543,-177.766,7.182,148.694
C05173=1165.675,217.120,-62.569,-177.763,7.185,148.694
C05174=1165.670,217.370,-62.594,-177.761,7.187,148.694
C05175=1165.665,217.618,-62.619,-177.758,7.190,148.694
C05176=1165.662,217.867,-62.644,-177.756,7.192,148.694
C05177=1165.657,218.115,-62.669,-177.752,7.195,148.693
C05178=1165.652,218.365,-62.694,-177.750,7.197,148.693
C05179=1165.647,218.613,-62.719,-177.747,7.199,148.693
C05180=1165.643,218.862,-62.744,-177.745,7.201,148.693
C05181=1165.639,219.110,-62.769,-177.741,7.204,148.692
C05182=1165.635,219.359,-62.795,-177.739,7.206,148.692
C05183=1165.629,219.607,-62.820,-177.736,7.209,148.692
C05184=1165.625,219.856,-62.845,-177.734,7.211,148.692
C05185=1165.621,220.106,-62.870,-177.731,7.213,148.692
C05186=1165.616,220.354,-62.896,-177.728,7.216,148.692
C05187=1165.612,220.602,-62.921,-177.726,7.218,148.691
C05188=1165.607,220.851,-62.946,-177.723,7.220,148.691
C05189=1165.603,221.100,-62.971,-177.720,7.223,148.691
C05190=1165.598,221.348,-62.997,-177.717,7.225,148.691
C05191=1165.594,221.597,-63.022,-177.715,7.228,148.691
C05192=1165.589,221.846,-63.048,-177.712,7.230,148.690
C05193=1165.585,222.094,-63.073,-177.709,7.233,148.690
C05194=1165.580,222.344,-63.098,-177.706,7.235,148.690
C05195=1165.575,222.592,-63.123,-177.704,7.237,148.690
C05196=1165.571,222.841,-63.149,-177.701,7.240,148.690
C05197=1165.567,223.089,-63.175,-177.698,7.242,148.689
C05198=1165.562,223.338,-63.200,-177.696,7.245,148.689
C05199=1165.557,223.587,-63.225,-177.693,7.247,148.689
C05200=1165.553,223.835,-63.251,-177.690,7.250,148.689
C05201=1165.549,224.083,-63.276,-177.688,7.252,148.688
C05202=1165.545,224.332,-63.302,-177.685,7.255,148.688
C05203=1165.540,224.580,-63.327,-177.682,7.257,148.688
C05204=1165.535,224.830,-63.353,-177.679,7.259,148.688
C05205=1165.531,225.079,-63.378,-177.677,7.262,148.688
C05206=1165.526,225.327,-63.404,-177.674,7.264,148.688
C05207=1165.522,225.576,-63.429,-177.671,7.267,148.687
C05208=1165.517,225.825,-63.455,-177.669,7.269,148.687
C05209=1165.512,226.073,-63.481,-177.666,7.272,148.687
C05210=1165.508,226.322,-63.506,-177.663,7.275,148.687
C05211=1165.504,226.570,-63.532,-177.660,7.276,148.687
C05212=1165.499,226.818,-63.557,-177.657,7.279,148.687
C05213=1165.495,227.067,-63.583,-177.655,7.281,148.686
C05214=1165.491,227.316,-63.609,-177.652,7.284,148.686
C05215=1165.486,227.564,-63.634,-177.650,7.286,148.686
C05216=1165.482,227.813,-63.660,-177.647,7.289,148.686
C05217=1165.477,228.062,-63.686,-177.644,7.292,148.686
C05218=1165.473,228.311,-63.712,-177.642,7.294,148.686
C05219=1165.468,228.559,-63.738,-177.638,7.296,148.685
C05220=1165.463,228.808,-63.763,-177.636,7.299,148.685
C05221=1165.459,229.057,-63.789,-177.633,7.302,148.685
C05222=1165.455,229.305,-63.815,-177.630,7.304,148.685
C05223=1165.450,229.553,-63.840,-177.628,7.306,148.685
C05224=1165.446,229.802,-63.866,-177.625,7.309,148.684
C05225=1165.441,230.051,-63.892,-177.623,7.311,148.684
C05226=1165.437,230.300,-63.918,-177.620,7.314,148.684
C05227=1165.432,230.548,-63.944,-177.617,7.317,148.684
C05228=1165.428,230.797,-63.970,-177.614,7.319,148.684
C05229=1165.424,231.045,-63.996,-177.612,7.322,148.684
C05230=1165.419,231.294,-64.022,-177.609,7.323,148.683
C05231=1165.415,231.543,-64.048,-177.606,7.326,148.683
C05232=1165.410,231.791,-64.073,-177.603,7.329,148.683
C05233=1165.406,232.040,-64.100,-177.601,7.331,148.683
C05234=1165.401,232.289,-64.126,-177.598,7.334,148.683
C05235=1165.397,232.537,-64.152,-177.595,7.337,148.683
C05236=1165.392,232.786,-64.177,-177.593,7.339,148.682
C05237=1165.387,233.034,-64.204,-177.590,7.342,148.682
C05238=1165.383,233.283,-64.230,-177.588,7.344,148.682
C05239=1165.379,233.532,-64.256,-177.584,7.346,148.682
C05240=1165.375,233.780,-64.281,-177.582,7.349,148.682
C05241=1165.370,234.029,-64.308,-177.579,7.352,148.682
C05242=1165.366,234.278,-64.334,-177.576,7.354,148.681
C05243=1165.361,234.526,-64.360,-177.573,7.357,148.681
C05244=1165.356,234.774,-64.387,-177.571,7.359,148.681
C05245=1165.352,235.023,-64.412,-177.568,7.362,148.681
C05246=1165.348,235.271,-64.439,-177.565,7.365,148.681
C05247=1165.343,235.520,-64.465,-177.563,7.367,148.681
C05248=1165.339,235.792,-64.494,-177.560,7.370,148.680
C05249=1165.333,236.064,-64.523,-177.557,7.372,148.680
C05250=1165.329,236.335,-64.551,-177.554,7.375,148.680
C05251=1165.323,236.607,-64.580,-177.551,7.378,148.680
C05252=1165.319,236.856,-64.607,-177.548,7.381,148.680
C05253=1165.315,237.104,-64.632,-177.546,7.383,148.680
C05254=1165.310,237.352,-64.659,-177.543,7.386,148.680
C05255=1165.306,237.601,-64.685,-177.540,7.389,148.679
C05256=1165.301,237.850,-64.712,-177.538,7.391,148.679
C05257=1165.297,238.098,-64.738,-177.535,7.393,148.679
C05258=1165.292,238.347,-64.765,-177.532,7.396,148.679
C05259=1165.288,238.596,-64.790,-177.530,7.399,148.679
C05260=1165.283,238.844,-64.817,-177.527,7.401,148.679
C05261=1165.279,239.093,-64.843,-177.524,7.404,148.679
C05262=1165.274,239.341,-64.870,-177.522,7.406,148.678
C05263=1165.271,239.590,-64.897,-177.519,7.409,148.678
C05264=1165.266,239.839,-64.923,-177.516,7.412,148.678
C05265=1165.262,240.087,-64.949,-177.513,7.415,148.678
C05266=1165.257,240.336,-64.976,-177.511,7.417,148.678
C05267=1165.253,240.584,-65.002,-177.508,7.420,148.678
C05268=1165.248,240.833,-65.029,-177.505,7.422,148.678
C05269=1165.244,241.082,-65.055,-177.502,7.425,148.677
C05270=1165.239,241.330,-65.082,-177.500,7.427,148.677
C05271=1165.235,241.578,-65.109,-177.497,7.430,148.677
C05272=1165.231,241.827,-65.136,-177.495,7.433,148.677
C05273=1165.226,242.076,-65.162,-177.491,7.435,148.677
C05274=1165.222,242.324,-65.189,-177.489,7.438,148.677
C05275=1165.217,242.573,-65.216,-177.487,7.440,148.677
C05276=1165.213,242.821,-65.242,-177.484,7.443,148.677
C05277=1165.208,243.070,-65.268,-177.481,7.446,148.676
C05278=1165.204,243.318,-65.295,-177.478,7.449,148.676
C05279=1165.200,243.566,-65.322,-177.476,7.451,148.676
C05280=1165.195,243.815,-65.349,-177.473,7.454,148.676
C05281=1165.190,244.063,-65.376,-177.470,7.456,148.676
C05282=1165.186,244.312,-65.402,-177.467,7.459,148.676
C05283=1165.182,244.561,-65.429,-177.465,7.462,148.676
C05284=1165.177,244.809,-65.456,-177.462,7.465,148.676
C05285=1165.173,245.057,-65.482,-177.460,7.467,148.675
C05286=1165.168,245.306,-65.509,-177.456,7.469,148.675
C05287=1165.164,245.554,-65.536,-177.454,7.472,148.675
C05288=1165.160,245.803,-65.563,-177.451,7.475,148.675
C05289=1165.156,246.052,-65.590,-177.449,7.477,148.675
C05290=1165.151,246.300,-65.617,-177.446,7.480,148.675
C05291=1165.146,246.549,-65.645,-177.443,7.483,148.675
C05292=1165.142,246.797,-65.671,-177.440,7.486,148.675
C05293=1165.138,247.045,-65.698,-177.438,7.488,148.674
C05294=1165.133,247.294,-65.725,-177.435,7.491,148.674
C05295=1165.128,247.542,-65.752,-177.432,7.494,148.674
C05296=1165.125,247.791,-65.779,-177.430,7.496,148.674
C05297=1165.120,248.039,-65.806,-177.427,7.499,148.674
C05298=1165.116,248.288,-65.833,-177.424,7.502,148.674
C05299=1165.111,248.537,-65.860,-177.421,7.505,148.674
C05300=1165.106,248.785,-65.887,-177.419,7.507,148.674
C05301=1165.103,249.034,-65.914,-177.416,7.510,148.674
C05302=1165.098,249.282,-65.941,-177.414,7.513,148.674
C05303=1165.093,249.531,-65.968,-177.410,7.515,148.673
C05304=1165.089,249.779,-65.995,-177.408,7.517,148.673
C05305=1165.085,250.028,-66.022,-177.405,7.520,148.673
C05306=1165.080,250.276,-66.050,-177.403,7.523,148.673
C05307=1165.076,250.525,-66.077,-177.400,7.526,148.673
C05308=1165.072,250.773,-66.104,-177.398,7.528,148.673
C05309=1165.067,251.021,-66.131,-177.395,7.531,148.673
C05310=1165.063,251.270,-66.158,-177.392,7.534,148.673
C05311=1165.059,251.518,-66.186,-177.389,7.537,148.672
C05312=1165.054,251.767,-66.213,-177.387,7.539,148.672
C05313=1165.049,252.015,-66.240,-177.384,7.542,148.672
C05314=1165.045,252.264,-66.267,-177.381,7.545,148.672
C05315=1165.041,252.512,-66.295,-177.379,7.548,148.672
C05316=1165.036,252.761,-66.322,-177.376,7.550,148.672
C05317=1165.032,253.009,-66.349,-177.374,7.553,148.672
C05318=1165.027,253.258,-66.376,-177.370,7.556,148.672
C05319=1165.023,253.506,-66.405,-177.368,7.558,148.672
C05320=1165.018,253.755,-66.432,-177.365,7.561,148.672
C05321=1165.014,254.003,-66.459,-177.363,7.564,148.672
C05322=1165.009,254.251,-66.486,-177.360,7.567,148.671
C05323=1165.005,254.501,-66.514,-177.357,7.569,148.671
C05324=1165.001,254.748,-66.542,-177.354,7.572,148.671
C05325=1164.996,254.997,-66.569,-177.352,7.575,148.671
C05326=1164.992,255.245,-66.596,-177.349,7.578,148.671
C05327=1164.988,255.494,-66.624,-177.347,7.580,148.671
C05328=1164.983,255.742,-66.651,-177.343,7.583,148.671
C05329=1164.979,255.990,-66.679,-177.341,7.586,148.671
C05330=1164.975,256.240,-66.706,-177.339,7.588,148.671
C05331=1164.971,256.487,-66.734,-177.336,7.591,148.671
C05332=1164.966,256.736,-66.761,-177.333,7.594,148.671
C05333=1164.962,256.985,-66.789,-177.330,7.597,148.671
C05334=1164.958,257.233,-66.816,-177.327,7.600,148.670
C05335=1164.953,257.481,-66.844,-177.325,7.602,148.670
C05336=1164.948,257.730,-66.872,-177.323,7.605,148.670
C05337=1164.944,257.978,-66.900,-177.320,7.608,148.670
C05338=1164.939,258.227,-66.927,-177.317,7.611,148.670
C05339=1164.936,258.475,-66.955,-177.314,7.614,148.670
C05340=1164.931,258.723,-66.983,-177.312,7.616,148.670
C05341=1164.927,258.972,-67.010,-177.309,7.619,148.670
C05342=1164.923,259.220,-67.038,-177.306,7.622,148.670
C05343=1164.917,259.469,-67.066,-177.303,7.625,148.670
C05344=1164.913,259.717,-67.093,-177.301,7.628,148.670
C05345=1164.909,259.966,-67.122,-177.298,7.630,148.669
C05346=1164.905,260.214,-67.149,-177.296,7.633,148.669
C05347=1164.901,260.463,-67.177,-177.293,7.636,148.669
C05348=1164.896,260.711,-67.205,-177.290,7.639,148.669
C05349=1164.892,260.959,-67.233,-177.287,7.642,148.669
C05350=1164.887,261.208,-67.260,-177.285,7.645,148.669
C05351=1164.883,261.456,-67.288,-177.282,7.647,148.669
C05352=1164.878,261.729,-67.319,-177.279,7.650,148.669
C05353=1164.874,262.002,-67.349,-177.276,7.653,148.669
C05354=1164.868,262.276,-67.381,-177.274,7.656,148.669
C05355=1164.863,262.549,-67.411,-177.271,7.659,148.669
C05356=1164.859,262.797,-67.439,-177.268,7.662,148.669
C05357=1164.855,263.045,-67.467,-177.265,7.665,148.669
C05358=1164.851,263.294,-67.496,-177.263,7.668,148.669
C05359=1164.846,263.542,-67.523,-177.260,7.671,148.669
C05360=1164.842,263.790,-67.552,-177.258,7.673,148.669
C05361=1164.837,264.039,-67.579,-177.255,7.676,148.669
C05362=1164.833,264.288,-67.607,-177.252,7.679,148.668
C05363=1164.829,264.536,-67.635,-177.249,7.682,148.668
C05364=1164.824,264.785,-67.664,-177.247,7.685,148.668
C05365=1164.820,265.032,-67.692,-177.244,7.688,148.668
C05366=1164.816,265.281,-67.720,-177.242,7.690,148.668
C05367=1164.811,265.529,-67.748,-177.239,7.693,148.668
C05368=1164.807,265.778,-67.776,-177.236,7.696,148.668
C05369=1164.802,266.026,-67.805,-177.233,7.699,148.668
C05370=1164.799,266.275,-67.833,-177.231,7.702,148.668
C05371=1164.794,266.522,-67.861,-177.228,7.705,148.668
C05372=1164.790,266.771,-67.889,-177.225,7.708,148.668
C05373=1164.785,267.019,-67.917,-177.223,7.710,148.668
C05374=1164.781,267.268,-67.946,-177.220,7.713,148.668
C05375=1164.777,267.516,-67.974,-177.217,7.716,148.668
C05376=1164.772,267.765,-68.002,-177.215,7.719,148.668
C05377=1164.768,268.013,-68.030,-177.212,7.722,148.668
C05378=1164.763,268.262,-68.059,-177.209,7.725,148.668
C05379=1164.759,268.510,-68.087,-177.206,7.728,148.668
C05380=1164.755,268.758,-68.116,-177.204,7.730,148.667
C05381=1164.751,269.006,-68.144,-177.201,7.733,148.667
C05382=1164.746,269.255,-68.173,-177.199,7.736,148.667
C05383=1164.742,269.503,-68.201,-177.196,7.739,148.667
C05384=1164.737,269.751,-68.229,-177.194,7.742,148.667
C05385=1164.733,270.000,-68.257,-177.191,7.745,148.667
C05386=1164.729,270.247,-68.286,-177.188,7.748,148.667
C05387=1164.725,270.496,-68.315,-177.185,7.751,148.667
C05388=1164.720,270.745,-68.343,-177.183,7.753,148.667
C05389=1164.716,270.993,-68.371,-177.180,7.756,148.667
C05390=1164.711,271.242,-68.400,-177.178,7.759,148.667
C05391=1164.707,271.490,-68.429,-177.175,7.762,148.667
C05392=1164.703,271.738,-68.457,-177.172,7.765,148.667
C05393=1164.698,271.987,-68.486,-177.169,7.768,148.667
C05394=1164.694,272.234,-68.514,-177.167,7.771,148.667
C05395=1164.690,272.483,-68.543,-177.164,7.774,148.667
C05396=1164.685,272.732,-68.572,-177.162,7.777,148.667
C05397=1164.681,272.979,-68.600,-177.159,7.779,148.667
C05398=1164.677,273.228,-68.629,-177.157,7.782,148.667
C05399=1164.672,273.477,-68.658,-177.154,7.785,148.667
C05400=1164.668,273.724,-68.686,-177.151,7.788,148.667
C05401=1164.664,273.973,-68.715,-177.148,7.791,148.667
C05402=1164.660,274.221,-68.744,-177.146,7.794,148.667
C05403=1164.655,274.469,-68.772,-177.143,7.797,148.667
C05404=1164.651,274.718,-68.801,-177.141,7.800,148.667
C05405=1164.647,274.966,-68.830,-177.138,7.803,148.667
C05406=1164.642,275.215,-68.859,-177.135,7.806,148.667
C05407=1164.638,275.462,-68.888,-177.132,7.809,148.667
C05408=1164.634,275.711,-68.916,-177.130,7.811,148.667
C05409=1164.629,275.960,-68.946,-177.127,7.814,148.667
C05410=1164.625,276.207,-68.974,-177.125,7.817,148.667
C05411=1164.621,276.456,-69.003,-177.122,7.820,148.666
C05412=1164.617,276.704,-69.032,-177.120,7.824,148.667
C05413=1164.612,276.953,-69.061,-177.117,7.826,148.667
C05414=1164.608,277.200,-69.090,-177.114,7.829,148.667
C05415=1164.604,277.449,-69.118,-177.111,7.832,148.666
C05416=1164.600,277.697,-69.148,-177.109,7.835,148.666
C05417=1164.595,277.946,-69.177,-177.106,7.838,148.666
C05418=1164.590,278.194,-69.206,-177.104,7.842,148.667
C05419=1164.586,278.442,-69.235,-177.101,7.845,148.667
C05420=1164.582,278.691,-69.263,-177.099,7.847,148.666
C05421=1164.578,278.939,-69.293,-177.096,7.850,148.666
C05422=1164.574,279.187,-69.322,-177.093,7.853,148.666
C05423=1164.569,279.435,-69.351,-177.090,7.856,148.666
C05424=1164.565,279.684,-69.380,-177.088,7.859,148.666
C05425=1164.561,279.932,-69.410,-177.085,7.862,148.666
C05426=1164.556,280.180,-69.439,-177.083,7.865,148.666
C05427=1164.553,280.429,-69.467,-177.080,7.868,148.666
C05428=1164.548,280.676,-69.496,-177.077,7.871,148.666
C05429=1164.544,280.924,-69.526,-177.075,7.874,148.666
C05430=1164.539,281.173,-69.555,-177.072,7.877,148.666
C05431=1164.535,281.422,-69.584,-177.069,7.880,148.666
C05432=1164.531,281.670,-69.613,-177.067,7.883,148.666
C05433=1164.527,281.918,-69.643,-177.064,7.886,148.666
C05434=1164.522,282.166,-69.672,-177.061,7.889,148.666
C05435=1164.518,282.414,-69.701,-177.059,7.892,148.666
C05436=1164.513,282.662,-69.731,-177.056,7.895,148.666
C05437=1164.509,282.911,-69.760,-177.054,7.897,148.666
C05438=1164.505,283.159,-69.789,-177.051,7.900,148.666
C05439=1164.501,283.408,-69.818,-177.049,7.903,148.666
C05440=1164.496,283.656,-69.848,-177.046,7.906,148.666
C05441=1164.492,283.903,-69.877,-177.043,7.909,148.666
C05442=1164.487,284.152,-69.906,-177.040,7.912,148.666
C05443=1164.483,284.400,-69.936,-177.038,7.916,148.667
C05444=1164.479,284.648,-69.965,-177.035,7.919,148.666
C05445=1164.475,284.897,-69.995,-177.033,7.922,148.666
C05446=1164.471,285.145,-70.024,-177.030,7.925,148.666
C05447=1164.467,285.393,-70.054,-177.027,7.928,148.666
C05448=1164.462,285.641,-70.083,-177.025,7.931,148.667
C05449=1164.457,285.890,-70.113,-177.022,7.934,148.666
C05450=1164.453,286.138,-70.143,-177.019,7.937,148.666
C05451=1164.449,286.386,-70.172,-177.017,7.940,148.666
C05452=1164.444,286.634,-70.201,-177.014,7.943,148.667
C05453=1164.440,286.882,-70.231,-177.012,7.946,148.667
C05454=1164.436,287.130,-70.261,-177.009,7.949,148.667
C05455=1164.432,287.378,-70.290,-177.007,7.952,148.667
C05456=1164.427,287.654,-70.323,-177.004,7.955,148.667
C05457=1164.423,287.928,-70.356,-177.000,7.959,148.667
C05458=1164.418,288.204,-70.389,-176.998,7.962,148.667
C05459=1164.413,288.479,-70.422,-176.995,7.965,148.667
C05460=1164.409,288.727,-70.452,-176.993,7.968,148.667
C05461=1164.405,288.975,-70.481,-176.990,7.971,148.667
C05462=1164.400,289.223,-70.510,-176.987,7.974,148.667
C05463=1164.397,289.471,-70.541,-176.984,7.977,148.667
C05464=1164.392,289.720,-70.571,-176.982,7.980,148.667
C05465=1164.387,289.968,-70.600,-176.979,7.983,148.667
C05466=1164.383,290.216,-70.630,-176.977,7.986,148.667
C05467=1164.379,290.464,-70.660,-176.974,7.990,148.667
C05468=1164.374,290.712,-70.690,-176.972,7.993,148.667
C05469=1164.370,290.961,-70.719,-176.969,7.995,148.667
C05470=1164.366,291.208,-70.749,-176.966,7.998,148.667
C05471=1164.362,291.456,-70.779,-176.964,8.002,148.667
C05472=1164.357,291.705,-70.809,-176.961,8.005,148.667
C05473=1164.353,291.953,-70.839,-176.958,8.008,148.667
C05474=1164.349,292.201,-70.869,-176.956,8.011,148.667
C05475=1164.344,292.450,-70.899,-176.953,8.014,148.667
C05476=1164.341,292.698,-70.929,-176.950,8.017,148.667
C05477=1164.337,292.946,-70.959,-176.948,8.020,148.667
C05478=1164.332,293.194,-70.989,-176.945,8.023,148.667
C05479=1164.328,293.442,-71.019,-176.943,8.026,148.667
C05480=1164.324,293.690,-71.049,-176.940,8.029,148.667
C05481=1164.319,293.939,-71.079,-176.938,8.032,148.667
C05482=1164.315,294.186,-71.109,-176.935,8.035,148.667
C05483=1164.311,294.435,-71.139,-176.933,8.039,148.667
C05484=1164.307,294.682,-71.169,-176.930,8.042,148.667
